// TIA Portal project "Traffic_Light" (V16)

(* hardware
DEVICE "S7-1200 station_1"  S7-1200 Station
   slot 0: "Rack_0"  S7-1200 Rack  Rack  V1.0
   slot 1: "PLC_1"  CPU 1214C DC/DC/DC  6ES7 214-1AG40-0XB0  V4.4
DEVICE "HMI_1"  KTP700 Basic PN
   slot 0: "HMI_1"  KTP700 Basic PN  6AV2 123-2GB03-0AX0  16.0.0.0
   slot 1: "HMI_RT_1"  KTP700 Basic PN  6AV2 123-2GB03-0AX0  16.0.0.0
   slot 5: "HMI_1.IE_CP_1"  PROFINET Interface  16.0.0.0
      slot 1: "PROFINET Interface_1"  PROFINET Interface
         slot 1: "Port_1"  Port
*)

// ===== PLC "PLC_1"  CPU 1214C DC/DC/DC =====

VAR_GLOBAL   // PLC tag table "Default tag table"
   "TrungGian" AT %M10.1 : Bool;
   "Clock_Byte" AT %MB0 : Byte;
   "Clock_10Hz" AT %M0.0 : Bool;
   "Clock_5Hz" AT %M0.1 : Bool;
   "Clock_2.5Hz" AT %M0.2 : Bool;
   "Clock_2Hz" AT %M0.3 : Bool;
   "Clock_1.25Hz" AT %M0.4 : Bool;
   "Clock_1Hz" AT %M0.5 : Bool;
   "Clock_0.625Hz" AT %M0.6 : Bool;
   "Clock_0.5Hz" AT %M0.7 : Bool;
   "Tag_1" AT %M20.1 : Bool;
END_VAR

DATA_BLOCK "DGT_DB"   // DB1
{ S7_Optimized_Access := 'TRUE' }
VERSION : 0.1
   VAR
      SP_TimerXA : Time := T#5S;
      SP_TimerVA : Time := T#3S;
      SP_TimerXB : Time := T#5S;
      SP_TimerVB : Time := T#3S;
      SP_TimerXA_PA4 : Int := 10;
      SP_TimerVA_PA4 : Int := 5;
      SP_TimerXB_PA4 : Int := 10;
      SP_TimerVB_PA4 : Int := 5;
      Lamp_PA1 : Bool;
      Lamp_PA2 : Bool;
      Lamp_PA4 : Bool;
      Update : Bool;
      Update_PA4 : Bool;
      Cancel : Bool;
      Temp_Update : Bool;
      Temp_Update_PA4 : Bool;
      Trunggian_Timer_1 : Bool;
      Trunggian_Timer_2 : Bool;
      OUT_XA : Bool;
      OUT_VA : Bool;
      OUT_DA : Bool;
      OUT_XB : Bool;
      OUT_VB : Bool;
      OUT_DB : Bool;
      OUT_XA_PA2 : Bool;
      OUT_VA_PA2 : Bool;
      OUT_DA_PA2 : Bool;
      OUT_XB_PA2 : Bool;
      OUT_VB_PA2 : Bool;
      OUT_DB_PA2 : Bool;
      OUT_XA_PA3 : Bool;
      OUT_VA_PA3 : Bool;
      OUT_DA_PA3 : Bool;
      OUT_XB_PA3 : Bool;
      OUT_VB_PA3 : Bool;
      OUT_DB_PA3 : Bool;
      OUT_XA_PA4 : Bool;
      OUT_VA_PA4 : Bool;
      OUT_DA_PA4 : Bool;
      OUT_XB_PA4 : Bool;
      OUT_VB_PA4 : Bool;
      OUT_DB_PA4 : Bool;
   END_VAR
BEGIN
END_DATA_BLOCK

DATA_BLOCK "DGT_TempVars"   // DB2
{ S7_Optimized_Access := 'TRUE' }
VERSION : 0.1
   VAR
      T1 : Time := T#5S;
      T2 : Time := T#8S;
      T3 : Time := T#13S;
      T4 : Time := T#16S;
      T1_PA4 : Int := 10;
      T2_PA4 : Int := 15;
      T3_PA4 : Int := 25;
      T4_PA4 : Int := 30;
      Temp : UInt;
      Temp_A : UInt;
      Temp_A_Chuc : UInt;
      Temp_A_DV : UInt;
      Temp_B : UInt;
      Temp_B_Chuc : UInt;
      Temp_B_DV : UInt;
      T11 : UInt;
      T22 : UInt;
      T33 : UInt;
      T44 : UInt;
      Temp_CK_PP1 : Time;
      Temp_SP_XA : Time := T#5S;
      Temp_SP_VA : Time := T#3S;
      Temp_SP_XB : Time := T#5S;
      Temp_SP_VB : Time := T#3S;
   END_VAR
BEGIN
END_DATA_BLOCK

DATA_BLOCK "Control"   // DB4
{ S7_Optimized_Access := 'TRUE' }
VERSION : 0.1
   VAR
      PA1_En : Bool;
      PA2_En : Bool;
      PA3_En : Bool;
      PA4_En : Bool;
      "ON/OFF_PP1" : Bool;
      "ON/OFF_PP2" : Bool;
      "ON/OFF_PP3" : Bool;
      "ON/OFF_PP4" : Bool;
      Stop : Bool;
   END_VAR
BEGIN
END_DATA_BLOCK

DATA_BLOCK "BCD_SEG_TEMPA_CHUC"   // DB10
{ S7_Optimized_Access := 'TRUE' }
VERSION : 0.1
// stored: InstanceOfName BCD_SEG
"BCD_SEG"
BEGIN
END_DATA_BLOCK

DATA_BLOCK "BCD_SEG_TEMPA_DV"   // DB11
{ S7_Optimized_Access := 'TRUE' }
VERSION : 0.1
// stored: InstanceOfName BCD_SEG
"BCD_SEG"
BEGIN
END_DATA_BLOCK

DATA_BLOCK "BCD_SEG_TEMPB_CHUC"   // DB12
{ S7_Optimized_Access := 'TRUE' }
VERSION : 0.1
// stored: InstanceOfName BCD_SEG
"BCD_SEG"
BEGIN
END_DATA_BLOCK

DATA_BLOCK "BCD_SEG_TEMPB_DV"   // DB13
{ S7_Optimized_Access := 'TRUE' }
VERSION : 0.1
// stored: InstanceOfName BCD_SEG
"BCD_SEG"
BEGIN
END_DATA_BLOCK

// folder: System blocks/Program resources

DATA_BLOCK "Timer_PP2"   // DB3
{ S7_Optimized_Access := 'TRUE' }
AUTHOR : Simatic
FAMILY : IEC
NAME : IEC_TMR
VERSION : 1.0
// stored: InstanceOfName IEC_TIMER
"IEC_TIMER"
BEGIN
END_DATA_BLOCK

DATA_BLOCK "T1_TIMER_PP1"   // DB5
{ S7_Optimized_Access := 'TRUE' }
AUTHOR : Simatic
FAMILY : IEC
NAME : IEC_TMR
VERSION : 1.0
// stored: InstanceOfName IEC_TIMER
"IEC_TIMER"
BEGIN
END_DATA_BLOCK

DATA_BLOCK "T2_TIMER_PP1"   // DB6
{ S7_Optimized_Access := 'TRUE' }
AUTHOR : Simatic
FAMILY : IEC
NAME : IEC_TMR
VERSION : 1.0
// stored: InstanceOfName IEC_TIMER
"IEC_TIMER"
BEGIN
END_DATA_BLOCK

DATA_BLOCK "T3_TIMER_PP1"   // DB7
{ S7_Optimized_Access := 'TRUE' }
AUTHOR : Simatic
FAMILY : IEC
NAME : IEC_TMR
VERSION : 1.0
// stored: InstanceOfName IEC_TIMER
"IEC_TIMER"
BEGIN
END_DATA_BLOCK

DATA_BLOCK "T4_TIMER_PP1"   // DB8
{ S7_Optimized_Access := 'TRUE' }
AUTHOR : Simatic
FAMILY : IEC
NAME : IEC_TMR
VERSION : 1.0
// stored: InstanceOfName IEC_TIMER
"IEC_TIMER"
BEGIN
END_DATA_BLOCK

DATA_BLOCK "Timer_PP1"   // DB9
{ S7_Optimized_Access := 'TRUE' }
AUTHOR : Simatic
FAMILY : IEC
NAME : IEC_TMR
VERSION : 1.0
// stored: InstanceOfName IEC_TIMER
"IEC_TIMER"
BEGIN
END_DATA_BLOCK

DATA_BLOCK "C1_PA4"   // DB14
{ S7_Optimized_Access := 'TRUE' }
AUTHOR : Simatic
FAMILY : IEC
NAME : CNTR
VERSION : 1.0
// stored: InstanceOfName IEC_COUNTER
"IEC_COUNTER"
BEGIN
END_DATA_BLOCK

// folder: (top level)

FUNCTION_BLOCK "BCD_SEG"   // FB1, SCL
{ S7_Optimized_Access := 'TRUE' }
VERSION : 0.1
   VAR_INPUT
      BCD : Int;
   END_VAR
   VAR_OUTPUT
      SEG : Byte;
   END_VAR
   VAR_TEMP
      tmp : Byte;
   END_VAR
BEGIN
   IF #BCD = 0 THEN
       // Statement section IF
       #tmp := 63;
   END_IF;
   IF #BCD = 1 THEN
       // Statement section IF
       #tmp := 6;
   END_IF;
   IF #BCD = 2 THEN
       // Statement section IF
       #tmp := 91;
   END_IF;
   IF #BCD = 3 THEN
       // Statement section IF
       #tmp := 79;
   END_IF;
   IF #BCD = 4 THEN
       // Statement section IF
       #tmp := 102;
   END_IF;
   IF #BCD = 5 THEN
       // Statement section IF
       #tmp := 109;
   END_IF;
   IF #BCD = 6 THEN
       // Statement section IF
       #tmp := 125;
   END_IF;
   IF #BCD = 7 THEN
       // Statement section IF
       #tmp := 7;
   END_IF;
   IF #BCD = 8 THEN
       // Statement section IF
       #tmp := 127;
   END_IF;
   IF #BCD = 9 THEN
       // Statement section IF
       #tmp := 111;
   END_IF;
   #SEG := #tmp;
END_FUNCTION_BLOCK

FUNCTION "PA2" : Void   // FC1, LAD
{ S7_Optimized_Access := 'TRUE' }
VERSION : 0.1
   VAR_INPUT
      EN_2 : Bool;
   END_VAR
   VAR_TEMP   // added for the SCL form of the ladder/FBD networks
      _w1 : Bool;
      _w2 : Bool;
   END_VAR
BEGIN

REGION Network 1: Update
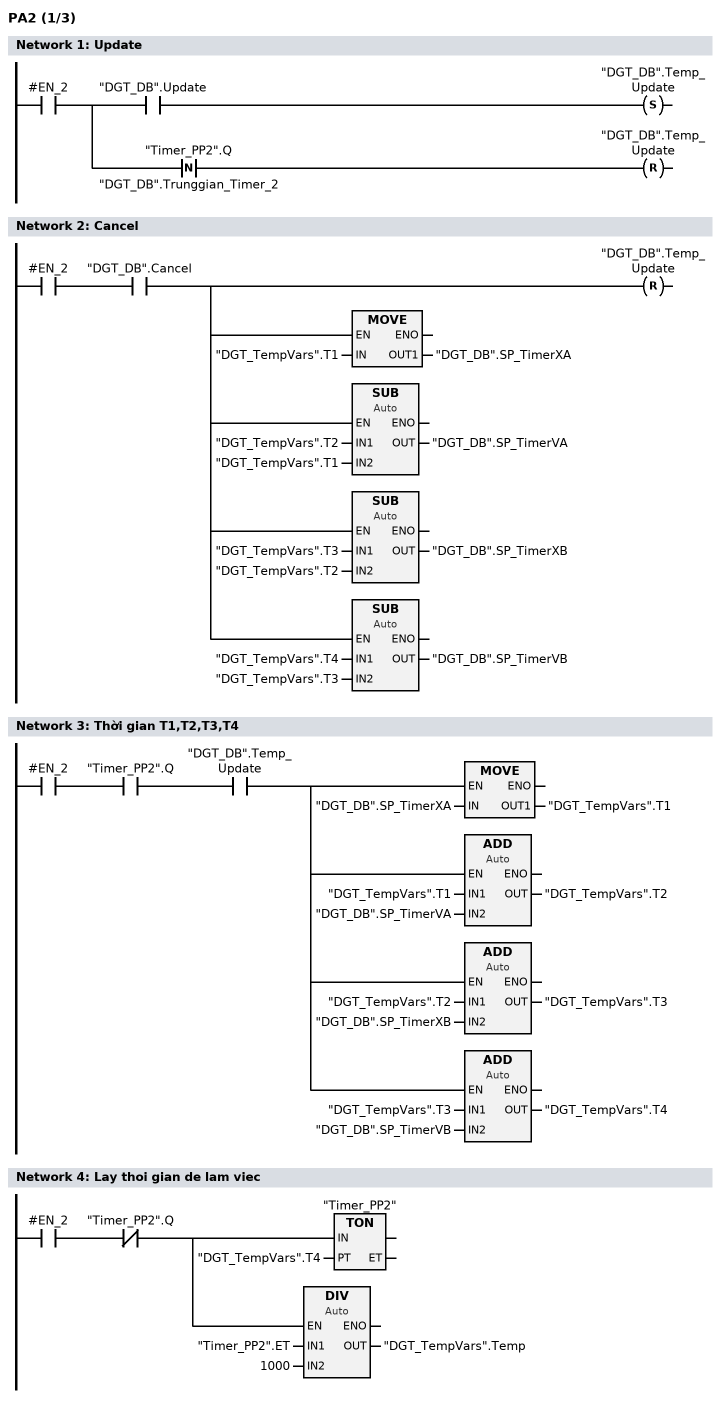
   RUNG wire#powerrail
      Contact( #EN_2 )
      wire#w1
      Contact( "DGT_DB".Update )
      S_Coil( "DGT_DB".Temp_Update )
   END_RUNG
   RUNG wire#w1
      N_Contact(operand := "Timer_PP2".Q, bit := "DGT_DB".Trunggian_Timer_2)
      R_Coil( "DGT_DB".Temp_Update )
   END_RUNG
   // the same network as SCL:
   IF #EN_2 AND "DGT_DB".Update THEN "DGT_DB".Temp_Update := TRUE; END_IF;
   #_w1 := #EN_2 AND NOT "Timer_PP2".Q AND "DGT_DB".Trunggian_Timer_2;   // falling edge of "Timer_PP2".Q
   "DGT_DB".Trunggian_Timer_2 := "Timer_PP2".Q;
   IF #_w1 THEN "DGT_DB".Temp_Update := FALSE; END_IF;
END_REGION

REGION Network 2: Cancel
   RUNG wire#powerrail
      Contact( #EN_2 )
      Contact( "DGT_DB".Cancel )
      wire#w1
      R_Coil( "DGT_DB".Temp_Update )
   END_RUNG
   RUNG wire#w1
      Move(in := "DGT_TempVars".T1, out1 => "DGT_DB".SP_TimerXA)
   END_RUNG
   RUNG wire#w1
      Sub(in1 := "DGT_TempVars".T2, in2 := "DGT_TempVars".T1, out => "DGT_DB".SP_TimerVA)
   END_RUNG
   RUNG wire#w1
      Sub(in1 := "DGT_TempVars".T3, in2 := "DGT_TempVars".T2, out => "DGT_DB".SP_TimerXB)
   END_RUNG
   RUNG wire#w1
      Sub(in1 := "DGT_TempVars".T4, in2 := "DGT_TempVars".T3, out => "DGT_DB".SP_TimerVB)
   END_RUNG
   // the same network as SCL:
   IF #EN_2 AND "DGT_DB".Cancel THEN
       "DGT_DB".Temp_Update := FALSE;
       "DGT_DB".SP_TimerXA := "DGT_TempVars".T1;
       "DGT_DB".SP_TimerVA := "DGT_TempVars".T2 - "DGT_TempVars".T1;
       "DGT_DB".SP_TimerXB := "DGT_TempVars".T3 - "DGT_TempVars".T2;
       "DGT_DB".SP_TimerVB := "DGT_TempVars".T4 - "DGT_TempVars".T3;
   END_IF;
END_REGION

REGION Network 3: Thời gian T1,T2,T3,T4
   RUNG wire#powerrail
      Contact( #EN_2 )
      Contact( "Timer_PP2".Q )
      Contact( "DGT_DB".Temp_Update )
      wire#w1
      Move(in := "DGT_DB".SP_TimerXA, out1 => "DGT_TempVars".T1)
   END_RUNG
   RUNG wire#w1
      Add(in1 := "DGT_TempVars".T1, in2 := "DGT_DB".SP_TimerVA, out => "DGT_TempVars".T2)
   END_RUNG
   RUNG wire#w1
      Add(in1 := "DGT_TempVars".T2, in2 := "DGT_DB".SP_TimerXB, out => "DGT_TempVars".T3)
   END_RUNG
   RUNG wire#w1
      Add(in1 := "DGT_TempVars".T3, in2 := "DGT_DB".SP_TimerVB, out => "DGT_TempVars".T4)
   END_RUNG
   // the same network as SCL:
   IF #EN_2 AND "Timer_PP2".Q AND "DGT_DB".Temp_Update THEN
       "DGT_TempVars".T1 := "DGT_DB".SP_TimerXA;
       "DGT_TempVars".T2 := "DGT_TempVars".T1 + "DGT_DB".SP_TimerVA;
       "DGT_TempVars".T3 := "DGT_TempVars".T2 + "DGT_DB".SP_TimerXB;
       "DGT_TempVars".T4 := "DGT_TempVars".T3 + "DGT_DB".SP_TimerVB;
   END_IF;
END_REGION

REGION Network 4: Lay thoi gian de lam viec
   #_w1 := #EN_2 AND NOT "Timer_PP2".Q;
   "Timer_PP2".TON(IN := #_w1, PT := "DGT_TempVars".T4);
   IF #_w1 THEN "DGT_TempVars".Temp := "Timer_PP2".ET / 1000; END_IF;
END_REGION

REGION Network 5: XA,VA,XB,VB
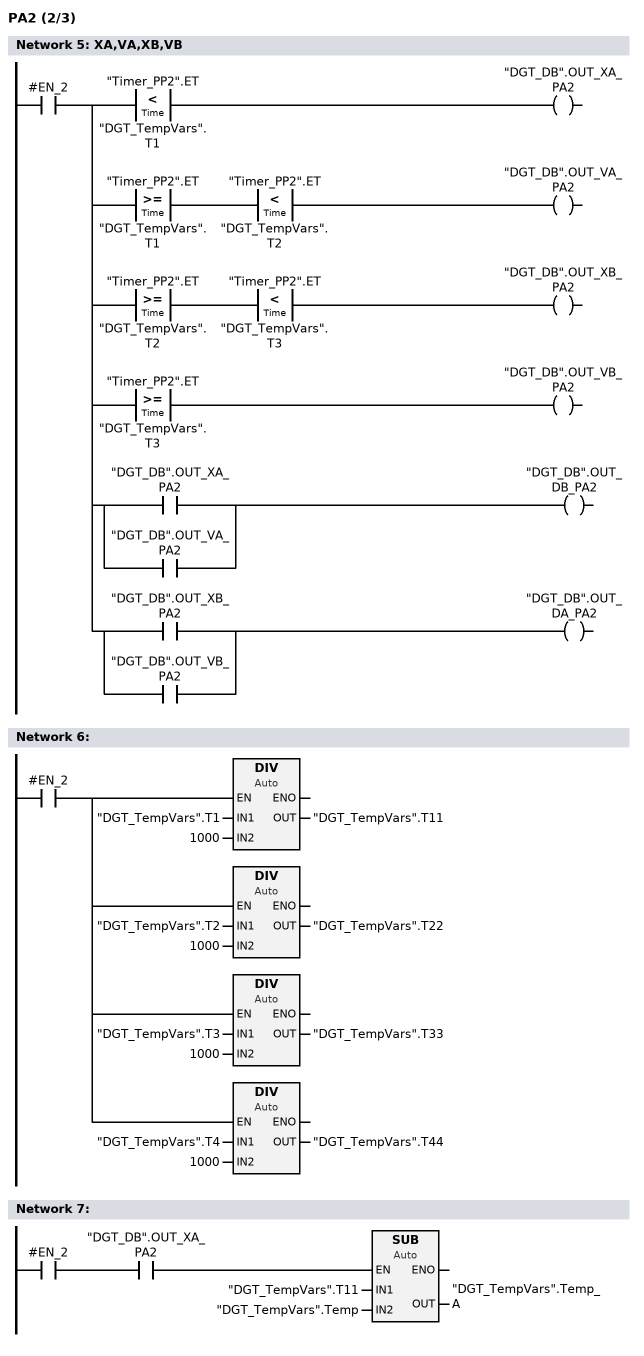
   RUNG wire#powerrail
      Contact( #EN_2 )
      wire#w1
      { S7_Templates := "SrcType := Time" } LT_Contact(in1 := "Timer_PP2".ET, in2 := "DGT_TempVars".T1)
      Coil( "DGT_DB".OUT_XA_PA2 )
   END_RUNG
   RUNG wire#w1
      { S7_Templates := "SrcType := Time" } GE_Contact(in1 := "Timer_PP2".ET, in2 := "DGT_TempVars".T1)
      { S7_Templates := "SrcType := Time" } LT_Contact(in1 := "Timer_PP2".ET, in2 := "DGT_TempVars".T2)
      Coil( "DGT_DB".OUT_VA_PA2 )
   END_RUNG
   RUNG wire#w1
      { S7_Templates := "SrcType := Time" } GE_Contact(in1 := "Timer_PP2".ET, in2 := "DGT_TempVars".T2)
      { S7_Templates := "SrcType := Time" } LT_Contact(in1 := "Timer_PP2".ET, in2 := "DGT_TempVars".T3)
      Coil( "DGT_DB".OUT_XB_PA2 )
   END_RUNG
   RUNG wire#w1
      { S7_Templates := "SrcType := Time" } GE_Contact(in1 := "Timer_PP2".ET, in2 := "DGT_TempVars".T3)
      Coil( "DGT_DB".OUT_VB_PA2 )
   END_RUNG
   RUNG wire#w1
      Contact( "DGT_DB".OUT_XA_PA2 )
      wire#w2
      Coil( "DGT_DB".OUT_DB_PA2 )
   END_RUNG
   RUNG wire#w1
      Contact( "DGT_DB".OUT_VA_PA2 )
   END_RUNG wire#w2
   RUNG wire#w1
      Contact( "DGT_DB".OUT_XB_PA2 )
      wire#w3
      Coil( "DGT_DB".OUT_DA_PA2 )
   END_RUNG
   RUNG wire#w1
      Contact( "DGT_DB".OUT_VB_PA2 )
   END_RUNG wire#w3
   // the same network as SCL:
   "DGT_DB".OUT_XA_PA2 := #EN_2 AND ("Timer_PP2".ET < "DGT_TempVars".T1);
   "DGT_DB".OUT_VA_PA2 := #EN_2 AND ("Timer_PP2".ET >= "DGT_TempVars".T1) AND ("Timer_PP2".ET < "DGT_TempVars".T2);
   "DGT_DB".OUT_XB_PA2 := #EN_2 AND ("Timer_PP2".ET >= "DGT_TempVars".T2) AND ("Timer_PP2".ET < "DGT_TempVars".T3);
   "DGT_DB".OUT_VB_PA2 := #EN_2 AND ("Timer_PP2".ET >= "DGT_TempVars".T3);
   "DGT_DB".OUT_DB_PA2 := #EN_2 AND ("DGT_DB".OUT_XA_PA2 OR "DGT_DB".OUT_VA_PA2);
   "DGT_DB".OUT_DA_PA2 := #EN_2 AND ("DGT_DB".OUT_XB_PA2 OR "DGT_DB".OUT_VB_PA2);
END_REGION

REGION Network 6
   RUNG wire#powerrail
      Contact( #EN_2 )
      wire#w1
      Div(in1 := "DGT_TempVars".T1, in2 := 1000, out => "DGT_TempVars".T11)
   END_RUNG
   RUNG wire#w1
      Div(in1 := "DGT_TempVars".T2, in2 := 1000, out => "DGT_TempVars".T22)
   END_RUNG
   RUNG wire#w1
      Div(in1 := "DGT_TempVars".T3, in2 := 1000, out => "DGT_TempVars".T33)
   END_RUNG
   RUNG wire#w1
      Div(in1 := "DGT_TempVars".T4, in2 := 1000, out => "DGT_TempVars".T44)
   END_RUNG
   // the same network as SCL:
   IF #EN_2 THEN
       "DGT_TempVars".T11 := "DGT_TempVars".T1 / 1000;
       "DGT_TempVars".T22 := "DGT_TempVars".T2 / 1000;
       "DGT_TempVars".T33 := "DGT_TempVars".T3 / 1000;
       "DGT_TempVars".T44 := "DGT_TempVars".T4 / 1000;
   END_IF;
END_REGION

REGION Network 7
   RUNG wire#powerrail
      Contact( #EN_2 )
      Contact( "DGT_DB".OUT_XA_PA2 )
      Sub(in1 := "DGT_TempVars".T11, in2 := "DGT_TempVars".Temp, out => "DGT_TempVars".Temp_A)
   END_RUNG
   // the same network as SCL:
   IF #EN_2 AND "DGT_DB".OUT_XA_PA2 THEN
       "DGT_TempVars".Temp_A := "DGT_TempVars".T11 - "DGT_TempVars".Temp;
   END_IF;
END_REGION

REGION Network 8
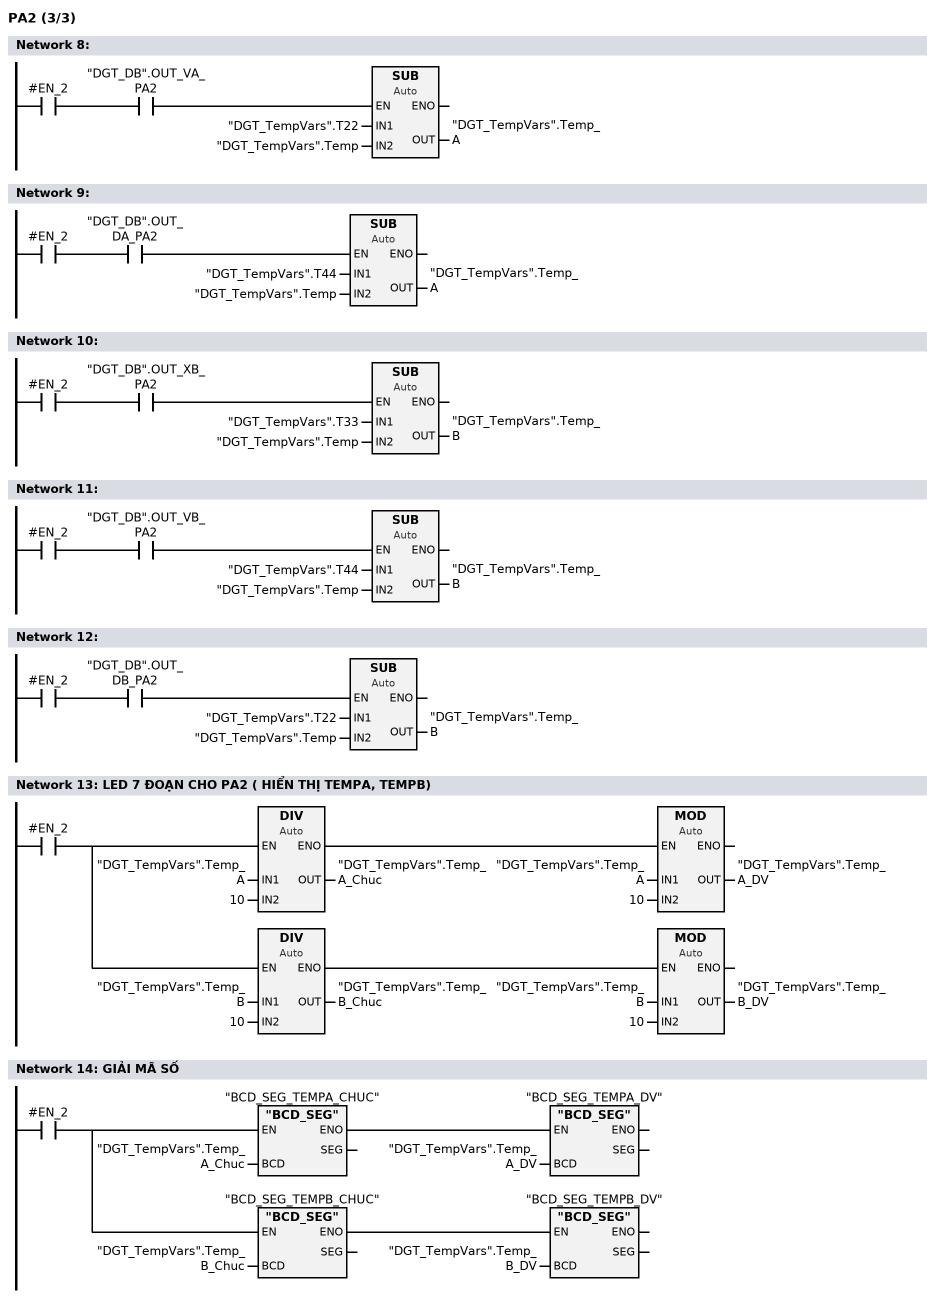
   RUNG wire#powerrail
      Contact( #EN_2 )
      Contact( "DGT_DB".OUT_VA_PA2 )
      Sub(in1 := "DGT_TempVars".T22, in2 := "DGT_TempVars".Temp, out => "DGT_TempVars".Temp_A)
   END_RUNG
   // the same network as SCL:
   IF #EN_2 AND "DGT_DB".OUT_VA_PA2 THEN
       "DGT_TempVars".Temp_A := "DGT_TempVars".T22 - "DGT_TempVars".Temp;
   END_IF;
END_REGION

REGION Network 9
   RUNG wire#powerrail
      Contact( #EN_2 )
      Contact( "DGT_DB".OUT_DA_PA2 )
      Sub(in1 := "DGT_TempVars".T44, in2 := "DGT_TempVars".Temp, out => "DGT_TempVars".Temp_A)
   END_RUNG
   // the same network as SCL:
   IF #EN_2 AND "DGT_DB".OUT_DA_PA2 THEN
       "DGT_TempVars".Temp_A := "DGT_TempVars".T44 - "DGT_TempVars".Temp;
   END_IF;
END_REGION

REGION Network 10
   RUNG wire#powerrail
      Contact( #EN_2 )
      Contact( "DGT_DB".OUT_XB_PA2 )
      Sub(in1 := "DGT_TempVars".T33, in2 := "DGT_TempVars".Temp, out => "DGT_TempVars".Temp_B)
   END_RUNG
   // the same network as SCL:
   IF #EN_2 AND "DGT_DB".OUT_XB_PA2 THEN
       "DGT_TempVars".Temp_B := "DGT_TempVars".T33 - "DGT_TempVars".Temp;
   END_IF;
END_REGION

REGION Network 11
   RUNG wire#powerrail
      Contact( #EN_2 )
      Contact( "DGT_DB".OUT_VB_PA2 )
      Sub(in1 := "DGT_TempVars".T44, in2 := "DGT_TempVars".Temp, out => "DGT_TempVars".Temp_B)
   END_RUNG
   // the same network as SCL:
   IF #EN_2 AND "DGT_DB".OUT_VB_PA2 THEN
       "DGT_TempVars".Temp_B := "DGT_TempVars".T44 - "DGT_TempVars".Temp;
   END_IF;
END_REGION

REGION Network 12
   RUNG wire#powerrail
      Contact( #EN_2 )
      Contact( "DGT_DB".OUT_DB_PA2 )
      Sub(in1 := "DGT_TempVars".T22, in2 := "DGT_TempVars".Temp, out => "DGT_TempVars".Temp_B)
   END_RUNG
   // the same network as SCL:
   IF #EN_2 AND "DGT_DB".OUT_DB_PA2 THEN
       "DGT_TempVars".Temp_B := "DGT_TempVars".T22 - "DGT_TempVars".Temp;
   END_IF;
END_REGION

REGION Network 13: LED 7 ĐOẠN CHO PA2 ( HIỂN THỊ TEMPA, TEMPB)
   RUNG wire#powerrail
      Contact( #EN_2 )
      wire#w1
      Div(in1 := "DGT_TempVars".Temp_A, in2 := 10, out => "DGT_TempVars".Temp_A_Chuc)
      Mod(in1 := "DGT_TempVars".Temp_A, in2 := 10, out => "DGT_TempVars".Temp_A_DV)
   END_RUNG
   RUNG wire#w1
      Div(in1 := "DGT_TempVars".Temp_B, in2 := 10, out => "DGT_TempVars".Temp_B_Chuc)
      Mod(in1 := "DGT_TempVars".Temp_B, in2 := 10, out => "DGT_TempVars".Temp_B_DV)
   END_RUNG
   // the same network as SCL:
   IF #EN_2 THEN
       "DGT_TempVars".Temp_A_Chuc := "DGT_TempVars".Temp_A / 10;
       "DGT_TempVars".Temp_A_DV := "DGT_TempVars".Temp_A MOD 10;
       "DGT_TempVars".Temp_B_Chuc := "DGT_TempVars".Temp_B / 10;
       "DGT_TempVars".Temp_B_DV := "DGT_TempVars".Temp_B MOD 10;
   END_IF;
END_REGION

REGION Network 14: GIẢI MÃ SỐ
   RUNG wire#powerrail
      Contact( #EN_2 )
      wire#w1
      "BCD_SEG_TEMPA_CHUC"(BCD := "DGT_TempVars".Temp_A_Chuc, SEG =>)
      "BCD_SEG_TEMPA_DV"(BCD := "DGT_TempVars".Temp_A_DV, SEG =>)
   END_RUNG
   RUNG wire#w1
      "BCD_SEG_TEMPB_CHUC"(BCD := "DGT_TempVars".Temp_B_Chuc, SEG =>)
      "BCD_SEG_TEMPB_DV"(BCD := "DGT_TempVars".Temp_B_DV, SEG =>)
   END_RUNG
   // the same network as SCL:
   "BCD_SEG_TEMPA_CHUC"(EN := #EN_2, BCD := "DGT_TempVars".Temp_A_Chuc, ENO => #_w1);   // "BCD_SEG"
   IF #_w1 THEN
       "BCD_SEG_TEMPA_DV"(BCD := "DGT_TempVars".Temp_A_DV);   // "BCD_SEG"
   END_IF;
   "BCD_SEG_TEMPB_CHUC"(EN := #EN_2, BCD := "DGT_TempVars".Temp_B_Chuc, ENO => #_w2);   // "BCD_SEG"
   IF #_w2 THEN
       "BCD_SEG_TEMPB_DV"(BCD := "DGT_TempVars".Temp_B_DV);   // "BCD_SEG"
   END_IF;
END_REGION
END_FUNCTION

FUNCTION "PA1" : Void   // FC2, LAD
{ S7_Optimized_Access := 'TRUE' }
VERSION : 0.1
   VAR_INPUT
      EN_1 : Bool;
   END_VAR
   VAR_TEMP   // added for the SCL form of the ladder/FBD networks
      _w1 : Bool;
      _w2 : Bool;
      _w3 : Bool;
   END_VAR
BEGIN

REGION Network 1: Update
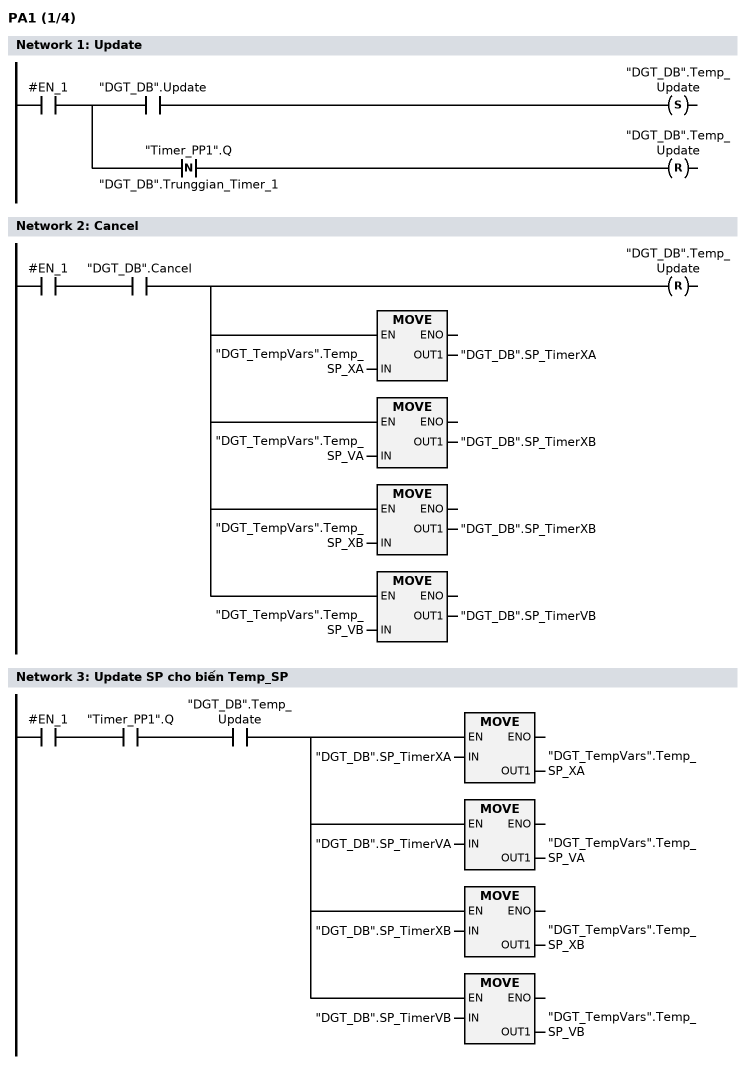
   RUNG wire#powerrail
      Contact( #EN_1 )
      wire#w1
      Contact( "DGT_DB".Update )
      S_Coil( "DGT_DB".Temp_Update )
   END_RUNG
   RUNG wire#w1
      N_Contact(operand := "Timer_PP1".Q, bit := "DGT_DB".Trunggian_Timer_1)
      R_Coil( "DGT_DB".Temp_Update )
   END_RUNG
   // the same network as SCL:
   IF #EN_1 AND "DGT_DB".Update THEN "DGT_DB".Temp_Update := TRUE; END_IF;
   #_w1 := #EN_1 AND NOT "Timer_PP1".Q AND "DGT_DB".Trunggian_Timer_1;   // falling edge of "Timer_PP1".Q
   "DGT_DB".Trunggian_Timer_1 := "Timer_PP1".Q;
   IF #_w1 THEN "DGT_DB".Temp_Update := FALSE; END_IF;
END_REGION

REGION Network 2: Cancel
   RUNG wire#powerrail
      Contact( #EN_1 )
      Contact( "DGT_DB".Cancel )
      wire#w1
      R_Coil( "DGT_DB".Temp_Update )
   END_RUNG
   RUNG wire#w1
      Move(in := "DGT_TempVars".Temp_SP_XA, out1 => "DGT_DB".SP_TimerXA)
   END_RUNG
   RUNG wire#w1
      Move(in := "DGT_TempVars".Temp_SP_VA, out1 => "DGT_DB".SP_TimerXB)
   END_RUNG
   RUNG wire#w1
      Move(in := "DGT_TempVars".Temp_SP_XB, out1 => "DGT_DB".SP_TimerXB)
   END_RUNG
   RUNG wire#w1
      Move(in := "DGT_TempVars".Temp_SP_VB, out1 => "DGT_DB".SP_TimerVB)
   END_RUNG
   // the same network as SCL:
   IF #EN_1 AND "DGT_DB".Cancel THEN
       "DGT_DB".Temp_Update := FALSE;
       "DGT_DB".SP_TimerXA := "DGT_TempVars".Temp_SP_XA;
       "DGT_DB".SP_TimerXB := "DGT_TempVars".Temp_SP_VA;
       "DGT_DB".SP_TimerXB := "DGT_TempVars".Temp_SP_XB;
       "DGT_DB".SP_TimerVB := "DGT_TempVars".Temp_SP_VB;
   END_IF;
END_REGION

REGION Network 3: Update SP cho biến Temp_SP
   RUNG wire#powerrail
      Contact( #EN_1 )
      Contact( "Timer_PP1".Q )
      Contact( "DGT_DB".Temp_Update )
      wire#w1
      Move(in := "DGT_DB".SP_TimerXA, out1 => "DGT_TempVars".Temp_SP_XA)
   END_RUNG
   RUNG wire#w1
      Move(in := "DGT_DB".SP_TimerVA, out1 => "DGT_TempVars".Temp_SP_VA)
   END_RUNG
   RUNG wire#w1
      Move(in := "DGT_DB".SP_TimerXB, out1 => "DGT_TempVars".Temp_SP_XB)
   END_RUNG
   RUNG wire#w1
      Move(in := "DGT_DB".SP_TimerVB, out1 => "DGT_TempVars".Temp_SP_VB)
   END_RUNG
   // the same network as SCL:
   IF #EN_1 AND "Timer_PP1".Q AND "DGT_DB".Temp_Update THEN
       "DGT_TempVars".Temp_SP_XA := "DGT_DB".SP_TimerXA;
       "DGT_TempVars".Temp_SP_VA := "DGT_DB".SP_TimerVA;
       "DGT_TempVars".Temp_SP_XB := "DGT_DB".SP_TimerXB;
       "DGT_TempVars".Temp_SP_VB := "DGT_DB".SP_TimerVB;
   END_IF;
END_REGION

REGION Network 4: Den Giao Thong
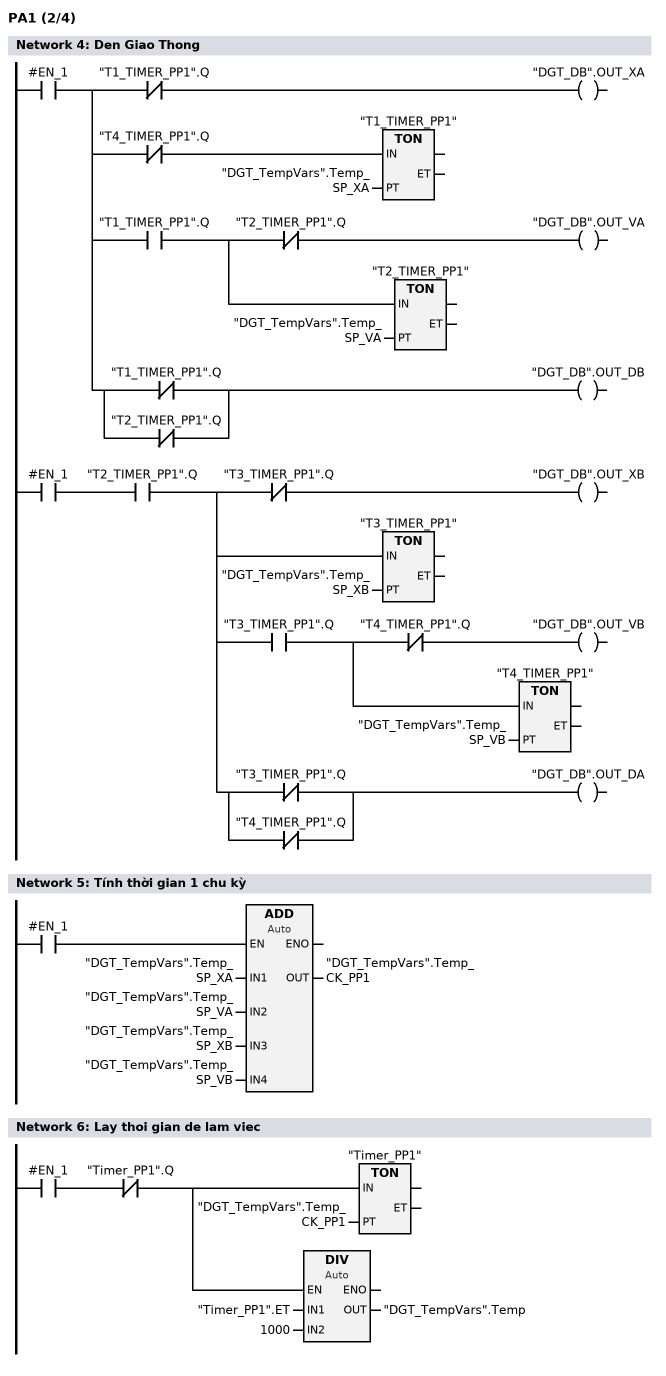
   "DGT_DB".OUT_XA := #EN_1 AND NOT "T1_TIMER_PP1".Q;
   "T1_TIMER_PP1".TON(IN := #EN_1 AND NOT "T4_TIMER_PP1".Q, PT := "DGT_TempVars".Temp_SP_XA);
   #_w1 := #EN_1 AND "T1_TIMER_PP1".Q;
   "DGT_DB".OUT_VA := #_w1 AND NOT "T2_TIMER_PP1".Q;
   "T2_TIMER_PP1".TON(IN := #_w1, PT := "DGT_TempVars".Temp_SP_VA);
   "DGT_DB".OUT_DB := #EN_1 AND (NOT "T1_TIMER_PP1".Q OR NOT "T2_TIMER_PP1".Q);
   #_w2 := #EN_1 AND "T2_TIMER_PP1".Q;
   "DGT_DB".OUT_XB := #_w2 AND NOT "T3_TIMER_PP1".Q;
   "T3_TIMER_PP1".TON(IN := #_w2, PT := "DGT_TempVars".Temp_SP_XB);
   #_w3 := #_w2 AND "T3_TIMER_PP1".Q;
   "DGT_DB".OUT_VB := #_w3 AND NOT "T4_TIMER_PP1".Q;
   "T4_TIMER_PP1".TON(IN := #_w3, PT := "DGT_TempVars".Temp_SP_VB);
   "DGT_DB".OUT_DA := #_w2 AND (NOT "T3_TIMER_PP1".Q OR NOT "T4_TIMER_PP1".Q);
END_REGION

REGION Network 5: Tính thời gian 1 chu kỳ
   RUNG wire#powerrail
      Contact( #EN_1 )
      Add(in1 := "DGT_TempVars".Temp_SP_XA, in2 := "DGT_TempVars".Temp_SP_VA, in3 := "DGT_TempVars".Temp_SP_XB, in4 := "DGT_TempVars".Temp_SP_VB, out => "DGT_TempVars".Temp_CK_PP1)
   END_RUNG
   // the same network as SCL:
   IF #EN_1 THEN
       "DGT_TempVars".Temp_CK_PP1 := "DGT_TempVars".Temp_SP_XA + "DGT_TempVars".Temp_SP_VA + "DGT_TempVars".Temp_SP_XB + "DGT_TempVars".Temp_SP_VB;
   END_IF;
END_REGION

REGION Network 6: Lay thoi gian de lam viec
   #_w1 := #EN_1 AND NOT "Timer_PP1".Q;
   "Timer_PP1".TON(IN := #_w1, PT := "DGT_TempVars".Temp_CK_PP1);
   IF #_w1 THEN "DGT_TempVars".Temp := "Timer_PP1".ET / 1000; END_IF;
END_REGION

REGION Network 7: Thời gian T1,T2,T3,T4
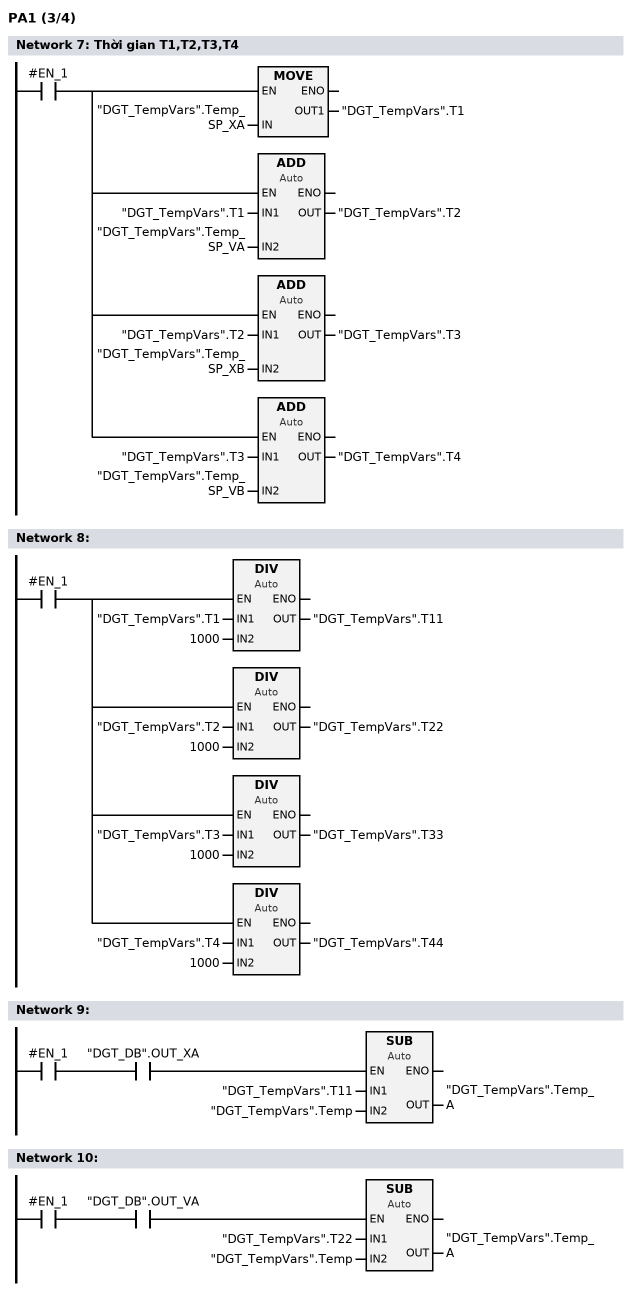
   RUNG wire#powerrail
      Contact( #EN_1 )
      wire#w1
      Move(in := "DGT_TempVars".Temp_SP_XA, out1 => "DGT_TempVars".T1)
   END_RUNG
   RUNG wire#w1
      Add(in1 := "DGT_TempVars".T1, in2 := "DGT_TempVars".Temp_SP_VA, out => "DGT_TempVars".T2)
   END_RUNG
   RUNG wire#w1
      Add(in1 := "DGT_TempVars".T2, in2 := "DGT_TempVars".Temp_SP_XB, out => "DGT_TempVars".T3)
   END_RUNG
   RUNG wire#w1
      Add(in1 := "DGT_TempVars".T3, in2 := "DGT_TempVars".Temp_SP_VB, out => "DGT_TempVars".T4)
   END_RUNG
   // the same network as SCL:
   IF #EN_1 THEN
       "DGT_TempVars".T1 := "DGT_TempVars".Temp_SP_XA;
       "DGT_TempVars".T2 := "DGT_TempVars".T1 + "DGT_TempVars".Temp_SP_VA;
       "DGT_TempVars".T3 := "DGT_TempVars".T2 + "DGT_TempVars".Temp_SP_XB;
       "DGT_TempVars".T4 := "DGT_TempVars".T3 + "DGT_TempVars".Temp_SP_VB;
   END_IF;
END_REGION

REGION Network 8
   RUNG wire#powerrail
      Contact( #EN_1 )
      wire#w1
      Div(in1 := "DGT_TempVars".T1, in2 := 1000, out => "DGT_TempVars".T11)
   END_RUNG
   RUNG wire#w1
      Div(in1 := "DGT_TempVars".T2, in2 := 1000, out => "DGT_TempVars".T22)
   END_RUNG
   RUNG wire#w1
      Div(in1 := "DGT_TempVars".T3, in2 := 1000, out => "DGT_TempVars".T33)
   END_RUNG
   RUNG wire#w1
      Div(in1 := "DGT_TempVars".T4, in2 := 1000, out => "DGT_TempVars".T44)
   END_RUNG
   // the same network as SCL:
   IF #EN_1 THEN
       "DGT_TempVars".T11 := "DGT_TempVars".T1 / 1000;
       "DGT_TempVars".T22 := "DGT_TempVars".T2 / 1000;
       "DGT_TempVars".T33 := "DGT_TempVars".T3 / 1000;
       "DGT_TempVars".T44 := "DGT_TempVars".T4 / 1000;
   END_IF;
END_REGION

REGION Network 9
   RUNG wire#powerrail
      Contact( #EN_1 )
      Contact( "DGT_DB".OUT_XA )
      Sub(in1 := "DGT_TempVars".T11, in2 := "DGT_TempVars".Temp, out => "DGT_TempVars".Temp_A)
   END_RUNG
   // the same network as SCL:
   IF #EN_1 AND "DGT_DB".OUT_XA THEN
       "DGT_TempVars".Temp_A := "DGT_TempVars".T11 - "DGT_TempVars".Temp;
   END_IF;
END_REGION

REGION Network 10
   RUNG wire#powerrail
      Contact( #EN_1 )
      Contact( "DGT_DB".OUT_VA )
      Sub(in1 := "DGT_TempVars".T22, in2 := "DGT_TempVars".Temp, out => "DGT_TempVars".Temp_A)
   END_RUNG
   // the same network as SCL:
   IF #EN_1 AND "DGT_DB".OUT_VA THEN
       "DGT_TempVars".Temp_A := "DGT_TempVars".T22 - "DGT_TempVars".Temp;
   END_IF;
END_REGION

REGION Network 11
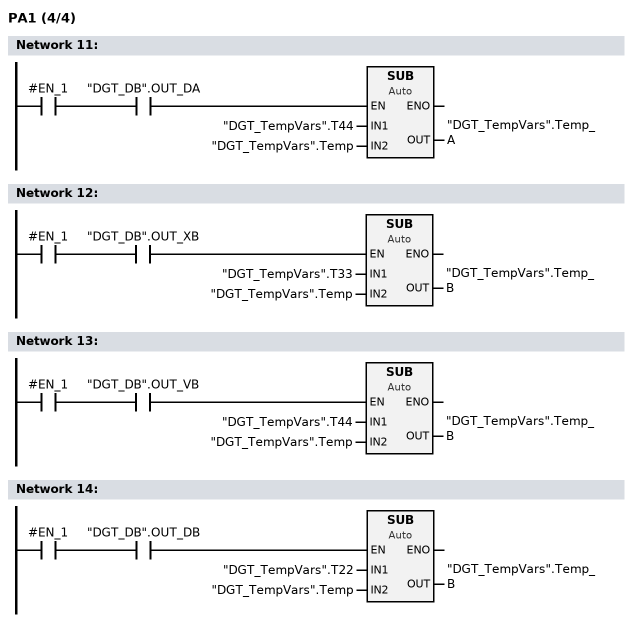
   RUNG wire#powerrail
      Contact( #EN_1 )
      Contact( "DGT_DB".OUT_DA )
      Sub(in1 := "DGT_TempVars".T44, in2 := "DGT_TempVars".Temp, out => "DGT_TempVars".Temp_A)
   END_RUNG
   // the same network as SCL:
   IF #EN_1 AND "DGT_DB".OUT_DA THEN
       "DGT_TempVars".Temp_A := "DGT_TempVars".T44 - "DGT_TempVars".Temp;
   END_IF;
END_REGION

REGION Network 12
   RUNG wire#powerrail
      Contact( #EN_1 )
      Contact( "DGT_DB".OUT_XB )
      Sub(in1 := "DGT_TempVars".T33, in2 := "DGT_TempVars".Temp, out => "DGT_TempVars".Temp_B)
   END_RUNG
   // the same network as SCL:
   IF #EN_1 AND "DGT_DB".OUT_XB THEN
       "DGT_TempVars".Temp_B := "DGT_TempVars".T33 - "DGT_TempVars".Temp;
   END_IF;
END_REGION

REGION Network 13
   RUNG wire#powerrail
      Contact( #EN_1 )
      Contact( "DGT_DB".OUT_VB )
      Sub(in1 := "DGT_TempVars".T44, in2 := "DGT_TempVars".Temp, out => "DGT_TempVars".Temp_B)
   END_RUNG
   // the same network as SCL:
   IF #EN_1 AND "DGT_DB".OUT_VB THEN
       "DGT_TempVars".Temp_B := "DGT_TempVars".T44 - "DGT_TempVars".Temp;
   END_IF;
END_REGION

REGION Network 14
   RUNG wire#powerrail
      Contact( #EN_1 )
      Contact( "DGT_DB".OUT_DB )
      Sub(in1 := "DGT_TempVars".T22, in2 := "DGT_TempVars".Temp, out => "DGT_TempVars".Temp_B)
   END_RUNG
   // the same network as SCL:
   IF #EN_1 AND "DGT_DB".OUT_DB THEN
       "DGT_TempVars".Temp_B := "DGT_TempVars".T22 - "DGT_TempVars".Temp;
   END_IF;
END_REGION
END_FUNCTION

FUNCTION "PA3" : Void   // FC3, LAD
{ S7_Optimized_Access := 'TRUE' }
VERSION : 0.1
BEGIN
END_FUNCTION

FUNCTION "PA4" : Void   // FC4, LAD
{ S7_Optimized_Access := 'TRUE' }
VERSION : 0.1
   VAR_INPUT
      EN_4 : Bool;
   END_VAR
   VAR_TEMP   // added for the SCL form of the ladder/FBD networks
      _w1 : Bool;
      _w2 : Bool;
   END_VAR
BEGIN

REGION Network 1
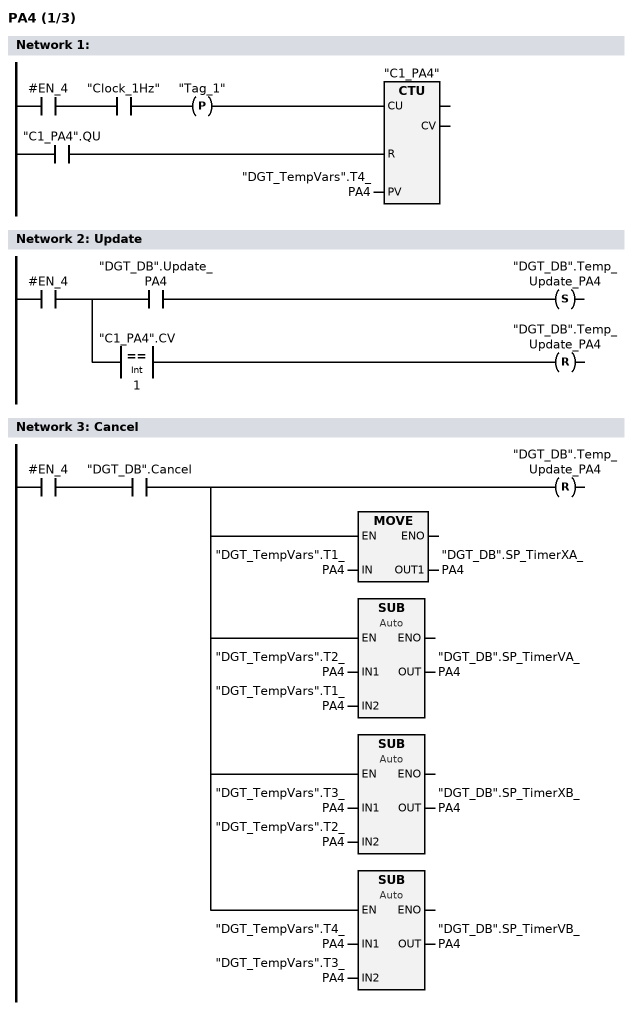
   #_w1 := #EN_4 AND "Clock_1Hz";
   #_w2 := #_w1 AND NOT "Tag_1";   // rising edge
   "Tag_1" := #_w1;
   "C1_PA4".CTU(CU := #_w2, R := "C1_PA4".QU, PV := "DGT_TempVars".T4_PA4);
END_REGION

REGION Network 2: Update
   RUNG wire#powerrail
      Contact( #EN_4 )
      wire#w1
      Contact( "DGT_DB".Update_PA4 )
      S_Coil( "DGT_DB".Temp_Update_PA4 )
   END_RUNG
   RUNG wire#w1
      { S7_Templates := "SrcType := Int" } EQ_Contact(in1 := "C1_PA4".CV, in2 := 1)
      R_Coil( "DGT_DB".Temp_Update_PA4 )
   END_RUNG
   // the same network as SCL:
   IF #EN_4 AND "DGT_DB".Update_PA4 THEN "DGT_DB".Temp_Update_PA4 := TRUE; END_IF;
   IF #EN_4 AND ("C1_PA4".CV = 1) THEN "DGT_DB".Temp_Update_PA4 := FALSE; END_IF;
END_REGION

REGION Network 3: Cancel
   RUNG wire#powerrail
      Contact( #EN_4 )
      Contact( "DGT_DB".Cancel )
      wire#w1
      R_Coil( "DGT_DB".Temp_Update_PA4 )
   END_RUNG
   RUNG wire#w1
      Move(in := "DGT_TempVars".T1_PA4, out1 => "DGT_DB".SP_TimerXA_PA4)
   END_RUNG
   RUNG wire#w1
      Sub(in1 := "DGT_TempVars".T2_PA4, in2 := "DGT_TempVars".T1_PA4, out => "DGT_DB".SP_TimerVA_PA4)
   END_RUNG
   RUNG wire#w1
      Sub(in1 := "DGT_TempVars".T3_PA4, in2 := "DGT_TempVars".T2_PA4, out => "DGT_DB".SP_TimerXB_PA4)
   END_RUNG
   RUNG wire#w1
      Sub(in1 := "DGT_TempVars".T4_PA4, in2 := "DGT_TempVars".T3_PA4, out => "DGT_DB".SP_TimerVB_PA4)
   END_RUNG
   // the same network as SCL:
   IF #EN_4 AND "DGT_DB".Cancel THEN
       "DGT_DB".Temp_Update_PA4 := FALSE;
       "DGT_DB".SP_TimerXA_PA4 := "DGT_TempVars".T1_PA4;
       "DGT_DB".SP_TimerVA_PA4 := "DGT_TempVars".T2_PA4 - "DGT_TempVars".T1_PA4;
       "DGT_DB".SP_TimerXB_PA4 := "DGT_TempVars".T3_PA4 - "DGT_TempVars".T2_PA4;
       "DGT_DB".SP_TimerVB_PA4 := "DGT_TempVars".T4_PA4 - "DGT_TempVars".T3_PA4;
   END_IF;
END_REGION

REGION Network 4: Thời gian T1,T2,T3,T4
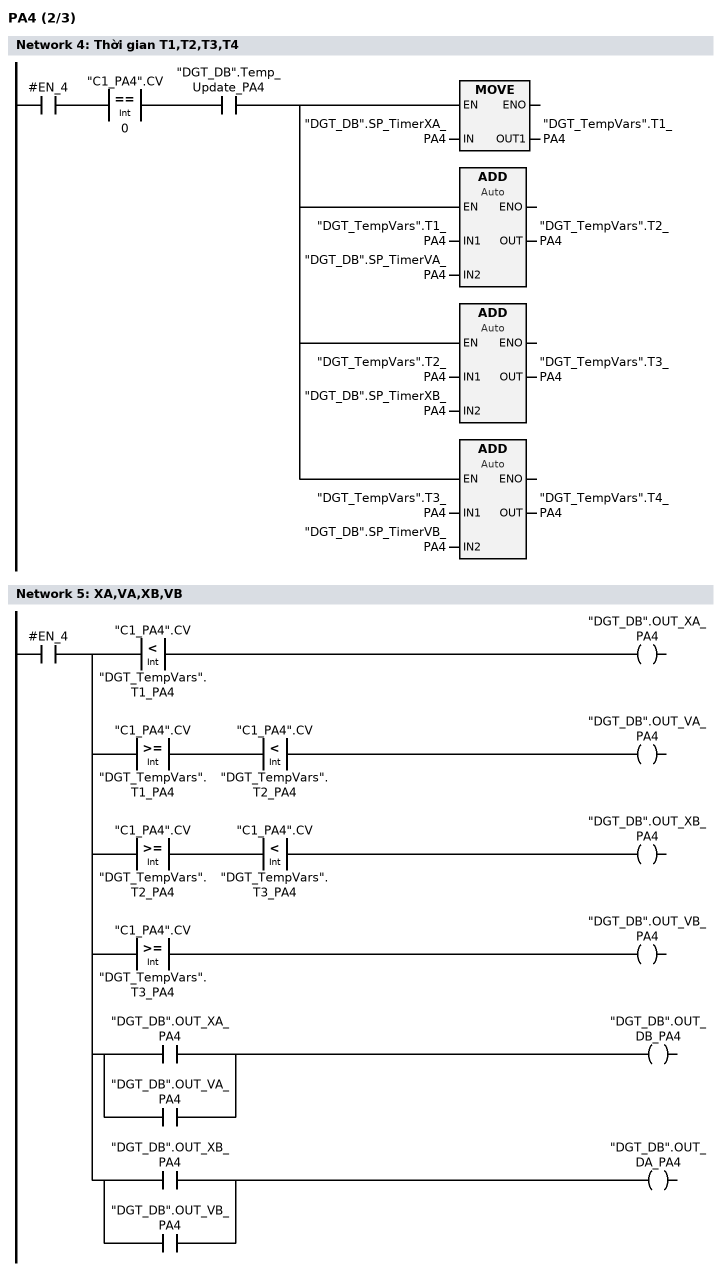
   RUNG wire#powerrail
      Contact( #EN_4 )
      { S7_Templates := "SrcType := Int" } EQ_Contact(in1 := "C1_PA4".CV, in2 := 0)
      Contact( "DGT_DB".Temp_Update_PA4 )
      wire#w1
      Move(in := "DGT_DB".SP_TimerXA_PA4, out1 => "DGT_TempVars".T1_PA4)
   END_RUNG
   RUNG wire#w1
      Add(in1 := "DGT_TempVars".T1_PA4, in2 := "DGT_DB".SP_TimerVA_PA4, out => "DGT_TempVars".T2_PA4)
   END_RUNG
   RUNG wire#w1
      Add(in1 := "DGT_TempVars".T2_PA4, in2 := "DGT_DB".SP_TimerXB_PA4, out => "DGT_TempVars".T3_PA4)
   END_RUNG
   RUNG wire#w1
      Add(in1 := "DGT_TempVars".T3_PA4, in2 := "DGT_DB".SP_TimerVB_PA4, out => "DGT_TempVars".T4_PA4)
   END_RUNG
   // the same network as SCL:
   IF #EN_4 AND ("C1_PA4".CV = 0) AND "DGT_DB".Temp_Update_PA4 THEN
       "DGT_TempVars".T1_PA4 := "DGT_DB".SP_TimerXA_PA4;
       "DGT_TempVars".T2_PA4 := "DGT_TempVars".T1_PA4 + "DGT_DB".SP_TimerVA_PA4;
       "DGT_TempVars".T3_PA4 := "DGT_TempVars".T2_PA4 + "DGT_DB".SP_TimerXB_PA4;
       "DGT_TempVars".T4_PA4 := "DGT_TempVars".T3_PA4 + "DGT_DB".SP_TimerVB_PA4;
   END_IF;
END_REGION

REGION Network 5: XA,VA,XB,VB
   RUNG wire#powerrail
      Contact( #EN_4 )
      wire#w1
      { S7_Templates := "SrcType := Int" } LT_Contact(in1 := "C1_PA4".CV, in2 := "DGT_TempVars".T1_PA4)
      Coil( "DGT_DB".OUT_XA_PA4 )
   END_RUNG
   RUNG wire#w1
      { S7_Templates := "SrcType := Int" } GE_Contact(in1 := "C1_PA4".CV, in2 := "DGT_TempVars".T1_PA4)
      { S7_Templates := "SrcType := Int" } LT_Contact(in1 := "C1_PA4".CV, in2 := "DGT_TempVars".T2_PA4)
      Coil( "DGT_DB".OUT_VA_PA4 )
   END_RUNG
   RUNG wire#w1
      { S7_Templates := "SrcType := Int" } GE_Contact(in1 := "C1_PA4".CV, in2 := "DGT_TempVars".T2_PA4)
      { S7_Templates := "SrcType := Int" } LT_Contact(in1 := "C1_PA4".CV, in2 := "DGT_TempVars".T3_PA4)
      Coil( "DGT_DB".OUT_XB_PA4 )
   END_RUNG
   RUNG wire#w1
      { S7_Templates := "SrcType := Int" } GE_Contact(in1 := "C1_PA4".CV, in2 := "DGT_TempVars".T3_PA4)
      Coil( "DGT_DB".OUT_VB_PA4 )
   END_RUNG
   RUNG wire#w1
      Contact( "DGT_DB".OUT_XA_PA4 )
      wire#w2
      Coil( "DGT_DB".OUT_DB_PA4 )
   END_RUNG
   RUNG wire#w1
      Contact( "DGT_DB".OUT_VA_PA4 )
   END_RUNG wire#w2
   RUNG wire#w1
      Contact( "DGT_DB".OUT_XB_PA4 )
      wire#w3
      Coil( "DGT_DB".OUT_DA_PA4 )
   END_RUNG
   RUNG wire#w1
      Contact( "DGT_DB".OUT_VB_PA4 )
   END_RUNG wire#w3
   // the same network as SCL:
   "DGT_DB".OUT_XA_PA4 := #EN_4 AND ("C1_PA4".CV < "DGT_TempVars".T1_PA4);
   "DGT_DB".OUT_VA_PA4 := #EN_4 AND ("C1_PA4".CV >= "DGT_TempVars".T1_PA4) AND ("C1_PA4".CV < "DGT_TempVars".T2_PA4);
   "DGT_DB".OUT_XB_PA4 := #EN_4 AND ("C1_PA4".CV >= "DGT_TempVars".T2_PA4) AND ("C1_PA4".CV < "DGT_TempVars".T3_PA4);
   "DGT_DB".OUT_VB_PA4 := #EN_4 AND ("C1_PA4".CV >= "DGT_TempVars".T3_PA4);
   "DGT_DB".OUT_DB_PA4 := #EN_4 AND ("DGT_DB".OUT_XA_PA4 OR "DGT_DB".OUT_VA_PA4);
   "DGT_DB".OUT_DA_PA4 := #EN_4 AND ("DGT_DB".OUT_XB_PA4 OR "DGT_DB".OUT_VB_PA4);
END_REGION

REGION Network 6
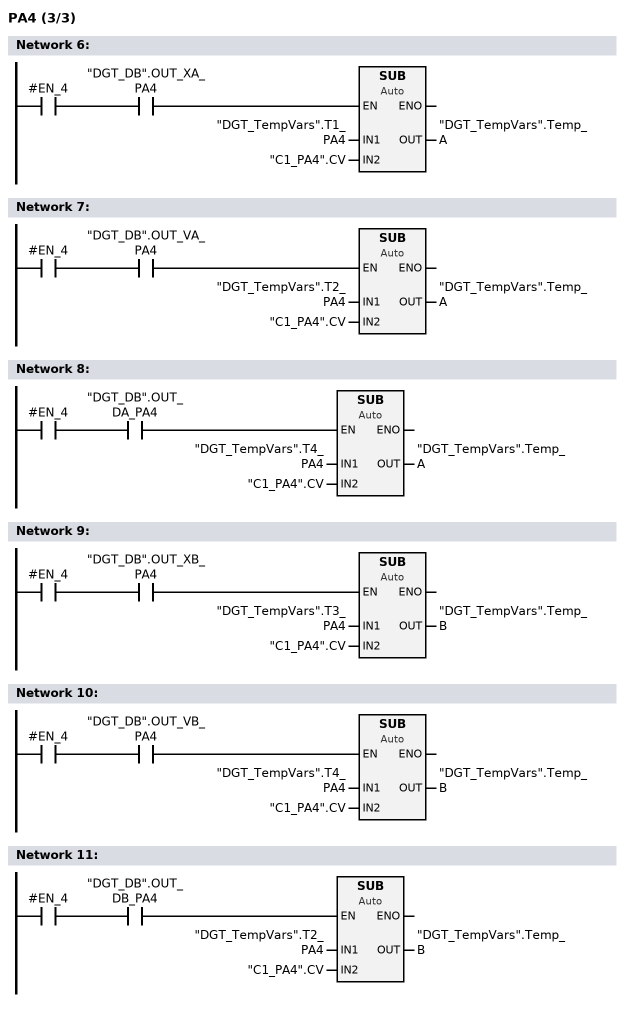
   RUNG wire#powerrail
      Contact( #EN_4 )
      Contact( "DGT_DB".OUT_XA_PA4 )
      Sub(in1 := "DGT_TempVars".T1_PA4, in2 := "C1_PA4".CV, out => "DGT_TempVars".Temp_A)
   END_RUNG
   // the same network as SCL:
   IF #EN_4 AND "DGT_DB".OUT_XA_PA4 THEN
       "DGT_TempVars".Temp_A := "DGT_TempVars".T1_PA4 - "C1_PA4".CV;
   END_IF;
END_REGION

REGION Network 7
   RUNG wire#powerrail
      Contact( #EN_4 )
      Contact( "DGT_DB".OUT_VA_PA4 )
      Sub(in1 := "DGT_TempVars".T2_PA4, in2 := "C1_PA4".CV, out => "DGT_TempVars".Temp_A)
   END_RUNG
   // the same network as SCL:
   IF #EN_4 AND "DGT_DB".OUT_VA_PA4 THEN
       "DGT_TempVars".Temp_A := "DGT_TempVars".T2_PA4 - "C1_PA4".CV;
   END_IF;
END_REGION

REGION Network 8
   RUNG wire#powerrail
      Contact( #EN_4 )
      Contact( "DGT_DB".OUT_DA_PA4 )
      Sub(in1 := "DGT_TempVars".T4_PA4, in2 := "C1_PA4".CV, out => "DGT_TempVars".Temp_A)
   END_RUNG
   // the same network as SCL:
   IF #EN_4 AND "DGT_DB".OUT_DA_PA4 THEN
       "DGT_TempVars".Temp_A := "DGT_TempVars".T4_PA4 - "C1_PA4".CV;
   END_IF;
END_REGION

REGION Network 9
   RUNG wire#powerrail
      Contact( #EN_4 )
      Contact( "DGT_DB".OUT_XB_PA4 )
      Sub(in1 := "DGT_TempVars".T3_PA4, in2 := "C1_PA4".CV, out => "DGT_TempVars".Temp_B)
   END_RUNG
   // the same network as SCL:
   IF #EN_4 AND "DGT_DB".OUT_XB_PA4 THEN
       "DGT_TempVars".Temp_B := "DGT_TempVars".T3_PA4 - "C1_PA4".CV;
   END_IF;
END_REGION

REGION Network 10
   RUNG wire#powerrail
      Contact( #EN_4 )
      Contact( "DGT_DB".OUT_VB_PA4 )
      Sub(in1 := "DGT_TempVars".T4_PA4, in2 := "C1_PA4".CV, out => "DGT_TempVars".Temp_B)
   END_RUNG
   // the same network as SCL:
   IF #EN_4 AND "DGT_DB".OUT_VB_PA4 THEN
       "DGT_TempVars".Temp_B := "DGT_TempVars".T4_PA4 - "C1_PA4".CV;
   END_IF;
END_REGION

REGION Network 11
   RUNG wire#powerrail
      Contact( #EN_4 )
      Contact( "DGT_DB".OUT_DB_PA4 )
      Sub(in1 := "DGT_TempVars".T2_PA4, in2 := "C1_PA4".CV, out => "DGT_TempVars".Temp_B)
   END_RUNG
   // the same network as SCL:
   IF #EN_4 AND "DGT_DB".OUT_DB_PA4 THEN
       "DGT_TempVars".Temp_B := "DGT_TempVars".T2_PA4 - "C1_PA4".CV;
   END_IF;
END_REGION
END_FUNCTION

ORGANIZATION_BLOCK "Main"   // OB1, LAD, ProgramCycle
TITLE = "Main Program Sweep (Cycle)"
{ S7_Optimized_Access := 'TRUE' }
VERSION : 0.1
   VAR_INPUT
      Initial_Call : Bool;   // Initial call of this OB
      Remanence : Bool;   // =True, if remanent data are available
   END_VAR
   VAR_TEMP   // added for the SCL form of the ladder/FBD networks
      _w1 : Bool;
   END_VAR
BEGIN

REGION Network 1
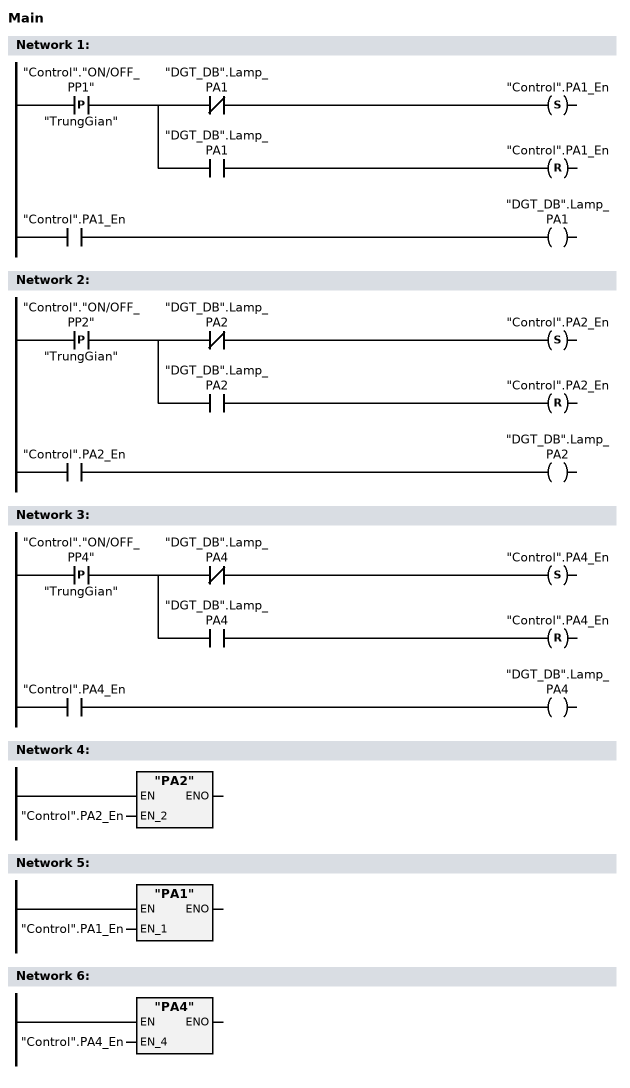
   RUNG wire#powerrail
      P_Contact(operand := "Control"."ON/OFF_PP1", bit := "TrungGian")
      wire#w1
      I_Contact( "DGT_DB".Lamp_PA1 )
      S_Coil( "Control".PA1_En )
   END_RUNG
   RUNG wire#w1
      Contact( "DGT_DB".Lamp_PA1 )
      R_Coil( "Control".PA1_En )
   END_RUNG
   RUNG wire#powerrail
      Contact( "Control".PA1_En )
      Coil( "DGT_DB".Lamp_PA1 )
   END_RUNG
   // the same network as SCL:
   #_w1 := "Control"."ON/OFF_PP1" AND NOT "TrungGian";   // rising edge of "Control"."ON/OFF_PP1"
   "TrungGian" := "Control"."ON/OFF_PP1";
   IF #_w1 AND NOT "DGT_DB".Lamp_PA1 THEN "Control".PA1_En := TRUE; END_IF;
   IF #_w1 AND "DGT_DB".Lamp_PA1 THEN "Control".PA1_En := FALSE; END_IF;
   "DGT_DB".Lamp_PA1 := "Control".PA1_En;
END_REGION

REGION Network 2
   RUNG wire#powerrail
      P_Contact(operand := "Control"."ON/OFF_PP2", bit := "TrungGian")
      wire#w1
      I_Contact( "DGT_DB".Lamp_PA2 )
      S_Coil( "Control".PA2_En )
   END_RUNG
   RUNG wire#w1
      Contact( "DGT_DB".Lamp_PA2 )
      R_Coil( "Control".PA2_En )
   END_RUNG
   RUNG wire#powerrail
      Contact( "Control".PA2_En )
      Coil( "DGT_DB".Lamp_PA2 )
   END_RUNG
   // the same network as SCL:
   #_w1 := "Control"."ON/OFF_PP2" AND NOT "TrungGian";   // rising edge of "Control"."ON/OFF_PP2"
   "TrungGian" := "Control"."ON/OFF_PP2";
   IF #_w1 AND NOT "DGT_DB".Lamp_PA2 THEN "Control".PA2_En := TRUE; END_IF;
   IF #_w1 AND "DGT_DB".Lamp_PA2 THEN "Control".PA2_En := FALSE; END_IF;
   "DGT_DB".Lamp_PA2 := "Control".PA2_En;
END_REGION

REGION Network 3
   RUNG wire#powerrail
      P_Contact(operand := "Control"."ON/OFF_PP4", bit := "TrungGian")
      wire#w1
      I_Contact( "DGT_DB".Lamp_PA4 )
      S_Coil( "Control".PA4_En )
   END_RUNG
   RUNG wire#w1
      Contact( "DGT_DB".Lamp_PA4 )
      R_Coil( "Control".PA4_En )
   END_RUNG
   RUNG wire#powerrail
      Contact( "Control".PA4_En )
      Coil( "DGT_DB".Lamp_PA4 )
   END_RUNG
   // the same network as SCL:
   #_w1 := "Control"."ON/OFF_PP4" AND NOT "TrungGian";   // rising edge of "Control"."ON/OFF_PP4"
   "TrungGian" := "Control"."ON/OFF_PP4";
   IF #_w1 AND NOT "DGT_DB".Lamp_PA4 THEN "Control".PA4_En := TRUE; END_IF;
   IF #_w1 AND "DGT_DB".Lamp_PA4 THEN "Control".PA4_En := FALSE; END_IF;
   "DGT_DB".Lamp_PA4 := "Control".PA4_En;
END_REGION

REGION Network 4
   RUNG wire#powerrail
      "PA2"(EN_2 := "Control".PA2_En)
   END_RUNG
   // the same network as SCL:
   "PA2"(EN_2 := "Control".PA2_En);
END_REGION

REGION Network 5
   RUNG wire#powerrail
      "PA1"(EN_1 := "Control".PA1_En)
   END_RUNG
   // the same network as SCL:
   "PA1"(EN_1 := "Control".PA1_En);
END_REGION

REGION Network 6
   RUNG wire#powerrail
      "PA4"(EN_4 := "Control".PA4_En)
   END_RUNG
   // the same network as SCL:
   "PA4"(EN_4 := "Control".PA4_En);
END_REGION
END_ORGANIZATION_BLOCK

(* ===== HMI "HMI_RT_1" =====
system functions are stored by id; their names below are inferred from use
connection "HMI_Connection_1": ETHERNET, SMART_S7_1200_OMS

HMI tags "Default tag table"
   "DGT_DB_SP_TimerXA" : Time = PLC DGT_DB.SP_TimerXA, 1 s
   "DGT_DB_SP_TimerVA" : Time = PLC DGT_DB.SP_TimerVA, 1 s
   "DGT_DB_SP_TimerXB" : Time = PLC DGT_DB.SP_TimerXB, 1 s
   "DGT_DB_SP_TimerVB" : Time = PLC DGT_DB.SP_TimerVB, 1 s
   "Timer_PP2_ET" : Time = PLC Timer_PP2.ET, 1 s
   "Control_PA2_En" : Bool = PLC Control.PA2_En, 1 s
   "Temp_A" : UInt = PLC DGT_TempVars.Temp_A AT %MD30, 1 s
   "Temp_B" : UInt = PLC DGT_TempVars.Temp_B AT %MD32, 1 s
   "DGT_TempVars_Temp_A" : UInt = PLC DGT_TempVars.Temp_A, 1 s
   "DGT_TempVars_Temp_B" : UInt = PLC DGT_TempVars.Temp_B, 1 s
   "DGT_TempVars_T1" : Time = PLC DGT_TempVars.T1, 1 s
   "DGT_TempVars_T2" : Time = PLC DGT_TempVars.T2, 1 s
   "DGT_TempVars_T3" : Time = PLC DGT_TempVars.T3, 1 s
   "DGT_TempVars_T4" : Time = PLC DGT_TempVars.T4, 1 s
   "DGT_DB_Lamp_PP2" : Bool = PLC DGT_DB.Lamp_PA2, 1 s
   "DGT_TempVars_Temp" : UInt = PLC DGT_TempVars.Temp, 1 s
   "DGT_DB_Update" : Bool = PLC DGT_DB.Update, 1 s
   "DGT_DB_Temp_Update" : Bool = PLC DGT_DB.Temp_Update, 1 s
   "DGT_DB_Cancel" : Bool = PLC DGT_DB.Cancel, 1 s
   "Control_PA1_En" : Bool = PLC Control.PA1_En, 1 s
   "DGT_TempVars_Temp_SP_XA" : Time = PLC DGT_TempVars.Temp_SP_XA, 1 s
   "DGT_TempVars_Temp_SP_VA" : Time = PLC DGT_TempVars.Temp_SP_VA, 1 s
   "DGT_TempVars_Temp_SP_XB" : Time = PLC DGT_TempVars.Temp_SP_XB, 1 s
   "DGT_TempVars_Temp_SP_VB" : Time = PLC DGT_TempVars.Temp_SP_VB, 1 s
   "Timer_PP1_ET" : Time = PLC Timer_PP1.ET, 1 s
   "DGT_DB_OUT_XA_PA2" : Bool = PLC DGT_DB.OUT_XA_PA2, 1 s
   "DGT_DB_OUT_VA_PA2" : Bool = PLC DGT_DB.OUT_VA_PA2, 1 s
   "DGT_DB_OUT_DA_PA2" : Bool = PLC DGT_DB.OUT_DA_PA2, 1 s
   "DGT_DB_OUT_XB_PA2" : Bool = PLC DGT_DB.OUT_XB_PA2, 1 s
   "DGT_DB_OUT_VB_PA2" : Bool = PLC DGT_DB.OUT_VB_PA2, 1 s
   "DGT_DB_OUT_DB_PA2" : Bool = PLC DGT_DB.OUT_DB_PA2, 1 s
   "DGT_DB_Lamp_PA1" : Bool = PLC DGT_DB.Lamp_PA1, 1 s
   "Control_ON/OFF_PP1" : Bool = PLC Control.ON/OFF_PP1, 1 s
   "Control_ON/OFF_PP2" : Bool = PLC Control.ON/OFF_PP2, 1 s
   "DGT_TempVars_T1_PA4" : Int = PLC DGT_TempVars.T1_PA4, 1 s
   "DGT_TempVars_T2_PA4" : Int = PLC DGT_TempVars.T2_PA4, 1 s
   "DGT_TempVars_T3_PA4" : Int = PLC DGT_TempVars.T3_PA4, 1 s
   "DGT_TempVars_T4_PA4" : Int = PLC DGT_TempVars.T4_PA4, 1 s
   "C1_PA4_CV" : Int = PLC C1_PA4.CV, 1 s
   "DGT_DB_OUT_XA_PA4" : Bool = PLC DGT_DB.OUT_XA_PA4, 1 s
   "DGT_DB_OUT_VA_PA4" : Bool = PLC DGT_DB.OUT_VA_PA4, 1 s
   "DGT_DB_OUT_DA_PA4" : Bool = PLC DGT_DB.OUT_DA_PA4, 1 s
   "DGT_DB_OUT_XB_PA4" : Bool = PLC DGT_DB.OUT_XB_PA4, 1 s
   "DGT_DB_OUT_VB_PA4" : Bool = PLC DGT_DB.OUT_VB_PA4, 1 s
   "DGT_DB_OUT_DB_PA4" : Bool = PLC DGT_DB.OUT_DB_PA4, 1 s
   "Control_ON/OFF_PP4" : Bool = PLC Control.ON/OFF_PP4, 1 s
   "DGT_DB_Lamp_PA4" : Bool = PLC DGT_DB.Lamp_PA4, 1 s
   "DGT_DB_SP_TimerXA_PA4" : Int = PLC DGT_DB.SP_TimerXA_PA4, 1 s
   "DGT_DB_SP_TimerVA_PA4" : Int = PLC DGT_DB.SP_TimerVA_PA4, 1 s
   "DGT_DB_SP_TimerXB_PA4" : Int = PLC DGT_DB.SP_TimerXB_PA4, 1 s
   "DGT_DB_SP_TimerVB_PA4" : Int = PLC DGT_DB.SP_TimerVB_PA4, 1 s
   "DGT_DB_Temp_Update_PA4" : Bool = PLC DGT_DB.Temp_Update_PA4, 1 s
   "DGT_DB_Update_PA4" : Bool = PLC DGT_DB.Update_PA4, 1 s
   "DGT_DB_OUT_XA" : Bool = PLC DGT_DB.OUT_XA, 1 s
   "DGT_DB_OUT_VA" : Bool = PLC DGT_DB.OUT_VA, 1 s
   "DGT_DB_OUT_DA" : Bool = PLC DGT_DB.OUT_DA, 1 s
   "DGT_DB_OUT_XB" : Bool = PLC DGT_DB.OUT_XB, 1 s
   "DGT_DB_OUT_VB" : Bool = PLC DGT_DB.OUT_VB, 1 s
   "DGT_DB_OUT_DB" : Bool = PLC DGT_DB.OUT_DB, 1 s
   "BCD_SEG_TEMPA_CHUC_SEG" : Byte = PLC BCD_SEG_TEMPA_CHUC.SEG, 1 s
   "BCD_SEG_TEMPA_DV_SEG" : Byte = PLC BCD_SEG_TEMPA_DV.SEG, 1 s
   "BCD_SEG_TEMPB_CHUC_SEG" : Byte = PLC BCD_SEG_TEMPB_CHUC.SEG, 1 s
   "BCD_SEG_TEMPB_DV_SEG" : Byte = PLC BCD_SEG_TEMPB_DV.SEG, 1 s

screen "Traffic_PA1" 800x480
   Circle "Circle_1" at 38,108 size 48x48
      Appearance <- "DGT_DB_OUT_DA"
   TextField "Text field_1" at 34,337 size 57x23; Text 'Side A'
   Circle "Circle_4" at 195,108 size 48x48
      Appearance <- "DGT_DB_OUT_DB"
   TextField "Text field_2" at 191,337 size 56x23; Text 'Side B'
   IOField "I/O field_6" at 23,36 size 83x41; FormatPattern 99
      ProcessValue <- "DGT_TempVars_Temp_A"
   IOField "I/O field_7" at 178,37 size 83x40; FormatPattern 99
      ProcessValue <- "DGT_TempVars_Temp_B"
   Circle "Circle_9" at 308,46 size 55x55
      Appearance <- "DGT_DB_Lamp_PA1"
   TextField "Text field_17" at 317,60 size 37x23; Text 'Run'
   Circle "Circle_10" at 308,106 size 55x55
      Appearance <- "DGT_DB_Temp_Update"
   TextField "Text field_19" at 309,122 size 51x20; Text 'Update'
   Button "Button_4" at 341,321 size 102x33; TextOff 'Start/Stop'
      on Press: SetBit("Control_ON/OFF_PP1")
      on Release: ResetBit("Control_ON/OFF_PP1")
   Button "Button_5" at 473,324 size 96x32; TextOff 'Update'
      on Release: ResetBit("DGT_DB_Update")
      on Press: SetBit("DGT_DB_Update")
   Button "Button_6" at 598,324 size 96x32; TextOff 'Cancel'
      on Release: ResetBit("DGT_DB_Cancel")
      on Press: SetBit("DGT_DB_Cancel")
   TextField "Text field_12" at 384,195 size 57x23; Text 'Side A'
   TextField "Text field_15" at 605,195 size 56x23; Text 'Side B'
   TextField "Text field_16" at 506,233 size 54x23; Text 'Green'
   TextField "Text field_20" at 506,271 size 60x23; Text 'Yellow'
   IOField "I/O field_12" at 366,225 size 107x32; FormatPattern s99999; Unit ms
      ProcessValue <- "DGT_DB_SP_TimerXA"
   IOField "I/O field_13" at 365,265 size 107x34; FormatPattern s99999; Unit ms
      ProcessValue <- "DGT_DB_SP_TimerVA"
   IOField "I/O field_14" at 569,223 size 114x36; FormatPattern s99999; Unit ms
      ProcessValue <- "DGT_DB_SP_TimerXB"
   IOField "I/O field_15" at 569,267 size 114x33; FormatPattern s99999; Unit ms
      ProcessValue <- "DGT_DB_SP_TimerVB"
   TextField "Text field_21" at 300,230 size 54x23; Text 'Green'
   TextField "Text field_22" at 300,270 size 60x23; Text 'Yellow'
   TextField "Text field_3" at 412,86 size 85x27; Text 'Running'
      Visibility <- "DGT_DB_Lamp_PA1"
   TextField "Text field_4" at 411,126 size 84x27; Text 'Stopped'
      Visibility <- "DGT_DB_Lamp_PA1"
   TextField "Text field_5" at 524,88 size 92x27; Text 'Updating'
      Visibility <- "DGT_DB_Temp_Update"
   TextField "Text field_7" at 523,127 size 85x27; Text 'Updated'
      Visibility <- "DGT_DB_Temp_Update"
   TextField "Text field_9" at 478,54 size 57x23; Text 'Status'
   IOField "I/O field_1" at 80,377 size 130x30; FormatPattern s9999999999
      ProcessValue <- "DGT_TempVars_Temp_SP_XA"
   IOField "I/O field_2" at 80,410 size 130x33; FormatPattern s9999999999
      ProcessValue <- "DGT_TempVars_Temp_SP_VA"
   IOField "I/O field_3" at 300,376 size 133x32; FormatPattern s9999999999
      ProcessValue <- "DGT_TempVars_Temp_SP_XB"
   IOField "I/O field_4" at 298,415 size 138x31; FormatPattern s9999999999
      ProcessValue <- "DGT_TempVars_Temp_SP_VB"
   IOField "I/O field_16" at 148,448 size 130x32; FormatPattern s9999999999
      ProcessValue <- "Timer_PP1_ET"
   TextField "Text field_6" at 261,7 size 286x27; Text 'Đèn Giao Thông Phương Án 1'
   Circle "Circle_2" at 38,246 size 48x48
      Appearance <- "DGT_DB_OUT_XA"
   Circle "Circle_3" at 38,175 size 48x48
      Appearance <- "DGT_DB_OUT_VA"
   Circle "Circle_5" at 193,240 size 48x48
      Appearance <- "DGT_DB_OUT_XB"
   Circle "Circle_6" at 193,175 size 48x48
      Appearance <- "DGT_DB_OUT_VB"
   TextField "Text field_8" at 113,453 size 26x23; Text 'ET'
   TextField "Text field_10" at 0,382 size 71x23; Text 'Green A'
   TextField "Text field_11" at 1,412 size 77x23; Text 'Yellow A'
   TextField "Text field_13" at 220,414 size 76x23; Text 'Yellow B'
   TextField "Text field_14" at 218,382 size 70x23; Text 'Green B'

screen "Traffic_PA2" 800x480
   Circle "Circle_1" at 39,151 size 48x48
      Appearance <- "DGT_DB_OUT_DA_PA2"
   Circle "Circle_2" at 39,217 size 48x48
      Appearance <- "DGT_DB_OUT_VA_PA2"
   Circle "Circle_3" at 39,284 size 48x48
      Appearance <- "DGT_DB_OUT_XA_PA2"
   TextField "Text field_1" at 35,344 size 57x23; Text 'Side A'
   Circle "Circle_4" at 196,148 size 48x48
      Appearance <- "DGT_DB_OUT_DB_PA2"
   Circle "Circle_5" at 196,214 size 48x48
      Appearance <- "DGT_DB_OUT_VB_PA2"
   Circle "Circle_6" at 196,281 size 48x48
      Appearance <- "DGT_DB_OUT_XB_PA2"
   TextField "Text field_2" at 192,344 size 56x23; Text 'Side B'
   IOField "I/O field_5" at 91,382 size 115x33; FormatPattern s99999; Unit ms
      ProcessValue <- "DGT_TempVars_T1"
   IOField "I/O field_8" at 93,415 size 113x34; FormatPattern s99999; Unit ms
      ProcessValue <- "DGT_TempVars_T2"
   IOField "I/O field_9" at 248,383 size 111x34; FormatPattern s99999; Unit ms
      ProcessValue <- "DGT_TempVars_T3"
   IOField "I/O field_10" at 248,417 size 112x31; FormatPattern s99999; Unit ms
      ProcessValue <- "DGT_TempVars_T4"
   IOField "I/O field_11" at 148,447 size 111x33; FormatPattern s99999; Unit ms
      ProcessValue <- "Timer_PP2_ET"
   TextField "Text field_6" at 56,386 size 26x23; Text 'T1'
   TextField "Text field_10" at 54,419 size 26x23; Text 'T2'
   TextField "Text field_11" at 222,386 size 26x23; Text 'T3'
   TextField "Text field_13" at 222,417 size 26x23; Text 'T4'
   TextField "Text field_14" at 107,449 size 26x23; Text 'ET'
   Circle "Circle_9" at 376,60 size 55x55
      Appearance <- "DGT_DB_Lamp_PP2"
   TextField "Text field_17" at 385,74 size 37x23; Text 'Run'
   Circle "Circle_10" at 376,120 size 55x55
      Appearance <- "DGT_DB_Temp_Update"
   TextField "Text field_19" at 377,136 size 51x20; Text 'Update'
   Button "Button_4" at 368,336 size 102x33; TextOff 'Start/Stop'
      on Release: ResetBit("Control_ON/OFF_PP2")
      on Press: SetBit("Control_ON/OFF_PP2")
   Button "Button_5" at 499,335 size 96x32; TextOff 'Update'
      on Release: ResetBit("DGT_DB_Update")
      on Press: SetBit("DGT_DB_Update")
   Button "Button_6" at 626,332 size 96x32; TextOff 'Cancel'
      on Release: ResetBit("DGT_DB_Cancel")
      on Press: SetBit("DGT_DB_Cancel")
   TextField "Text field_12" at 411,210 size 57x23; Text 'Side A'
   TextField "Text field_15" at 632,210 size 56x23; Text 'Side B'
   TextField "Text field_16" at 533,248 size 54x23; Text 'Green'
   TextField "Text field_20" at 533,286 size 60x23; Text 'Yellow'
   IOField "I/O field_12" at 393,240 size 107x32; FormatPattern s9999; Unit giây
      ProcessValue <- "DGT_DB_SP_TimerXA"
   IOField "I/O field_13" at 392,280 size 107x34; FormatPattern s9999; Unit giây
      ProcessValue <- "DGT_DB_SP_TimerVA"
   IOField "I/O field_14" at 596,238 size 114x36; FormatPattern s9999; Unit giây
      ProcessValue <- "DGT_DB_SP_TimerXB"
   IOField "I/O field_15" at 596,282 size 114x33; FormatPattern s9999; Unit giây
      ProcessValue <- "DGT_DB_SP_TimerVB"
   TextField "Text field_21" at 327,245 size 54x23; Text 'Green'
   TextField "Text field_22" at 327,285 size 60x23; Text 'Yellow'
   TextField "Text field_3" at 480,100 size 85x27; Text 'Running'
      Visibility <- "DGT_DB_Lamp_PP2"
   TextField "Text field_4" at 479,140 size 84x27; Text 'Stopped'
      Visibility <- "DGT_DB_Lamp_PP2"
   TextField "Text field_5" at 592,102 size 92x27; Text 'Updating'
      Visibility <- "DGT_DB_Temp_Update"
   TextField "Text field_7" at 591,141 size 85x27; Text 'Updated'
      Visibility <- "DGT_DB_Temp_Update"
   TextField "Text field_9" at 546,68 size 57x23; Text 'Status'
   TextField "Text field_18" at 9,405 size 36x23; Text 'PLC'
   Group "Group" at 16,34 size 100x93
   Group "Group_1" at 170,34 size 106x92
   TextField "Text field_23" at 387,12 size 250x27; Text 'Lập trình Đèn Giao Thông'
   Rectangle "Rectangle_7" at 21,34 size 38x8
      Appearance <- "BCD_SEG_TEMPA_CHUC_SEG"
   Rectangle "Rectangle_9" at 55,42 size 8x35
      Appearance <- "BCD_SEG_TEMPA_CHUC_SEG"
   Rectangle "Rectangle_10" at 16,42 size 8x35
      Appearance <- "BCD_SEG_TEMPA_CHUC_SEG"
   Rectangle "Rectangle_11" at 20,77 size 38x8
      Appearance <- "BCD_SEG_TEMPA_CHUC_SEG"
   Rectangle "Rectangle_12" at 54,84 size 8x35
      Appearance <- "BCD_SEG_TEMPA_CHUC_SEG"
   Rectangle "Rectangle_13" at 16,84 size 8x35
      Appearance <- "BCD_SEG_TEMPA_CHUC_SEG"
   Rectangle "Rectangle_14" at 21,119 size 38x8
      Appearance <- "BCD_SEG_TEMPA_CHUC_SEG"
   Rectangle "Rectangle_15" at 75,34 size 38x8
      Appearance <- "BCD_SEG_TEMPA_DV_SEG"
   Rectangle "Rectangle_16" at 108,42 size 8x35
      Appearance <- "BCD_SEG_TEMPA_DV_SEG"
   Rectangle "Rectangle_17" at 70,42 size 8x35
      Appearance <- "BCD_SEG_TEMPA_DV_SEG"
   Rectangle "Rectangle_18" at 74,77 size 38x8
      Appearance <- "BCD_SEG_TEMPA_DV_SEG"
   Rectangle "Rectangle_19" at 107,84 size 8x35
      Appearance <- "BCD_SEG_TEMPA_DV_SEG"
   Rectangle "Rectangle_20" at 70,84 size 8x35
      Appearance <- "BCD_SEG_TEMPA_DV_SEG"
   Rectangle "Rectangle_21" at 75,119 size 38x8
      Appearance <- "BCD_SEG_TEMPA_DV_SEG"
   Rectangle "Rectangle_22" at 175,34 size 40x8
      Appearance <- "BCD_SEG_TEMPB_CHUC_SEG"
   Rectangle "Rectangle_23" at 211,42 size 8x34
      Appearance <- "BCD_SEG_TEMPB_CHUC_SEG"
   Rectangle "Rectangle_24" at 170,42 size 8x34
      Appearance <- "BCD_SEG_TEMPB_CHUC_SEG"
   Rectangle "Rectangle_25" at 175,76 size 40x8
      Appearance <- "BCD_SEG_TEMPB_CHUC_SEG"
   Rectangle "Rectangle_26" at 210,84 size 8x34
      Appearance <- "BCD_SEG_TEMPB_CHUC_SEG"
   Rectangle "Rectangle_27" at 170,84 size 8x34
      Appearance <- "BCD_SEG_TEMPB_CHUC_SEG"
   Rectangle "Rectangle_28" at 175,118 size 40x8
      Appearance <- "BCD_SEG_TEMPB_CHUC_SEG"
   Rectangle "Rectangle_29" at 232,34 size 40x8
      Appearance <- "BCD_SEG_TEMPB_DV_SEG"
   Rectangle "Rectangle_30" at 268,42 size 8x34
      Appearance <- "BCD_SEG_TEMPB_DV_SEG"
   Rectangle "Rectangle_31" at 226,42 size 8x34
      Appearance <- "BCD_SEG_TEMPB_DV_SEG"
   Rectangle "Rectangle_32" at 231,76 size 40x8
      Appearance <- "BCD_SEG_TEMPB_DV_SEG"
   Rectangle "Rectangle_33" at 267,84 size 8x34
      Appearance <- "BCD_SEG_TEMPB_DV_SEG"
   Rectangle "Rectangle_34" at 226,84 size 8x34
      Appearance <- "BCD_SEG_TEMPB_DV_SEG"
   Rectangle "Rectangle_35" at 232,118 size 40x8
      Appearance <- "BCD_SEG_TEMPB_DV_SEG"

screen "Traffic_PA4" 800x480
   Circle "Circle_1" at 36,89 size 48x48
      Appearance <- "DGT_DB_OUT_DA_PA4"
   Circle "Circle_2" at 36,155 size 48x48
      Appearance <- "DGT_DB_OUT_VA_PA4"
   Circle "Circle_3" at 36,222 size 48x48
      Appearance <- "DGT_DB_OUT_XA_PA4"
   TextField "Text field_1" at 32,318 size 57x23; Text 'Side A'
   Circle "Circle_4" at 193,89 size 48x48
      Appearance <- "DGT_DB_OUT_DB_PA4"
   Circle "Circle_5" at 193,155 size 48x48
      Appearance <- "DGT_DB_OUT_VB_PA4"
   Circle "Circle_6" at 193,222 size 48x48
      Appearance <- "DGT_DB_OUT_XB_PA4"
   TextField "Text field_2" at 189,318 size 56x23; Text 'Side B'
   IOField "I/O field_6" at 21,17 size 83x41; FormatPattern 99
      ProcessValue <- "DGT_TempVars_Temp_A"
   IOField "I/O field_7" at 176,18 size 83x40; FormatPattern 99
      ProcessValue <- "DGT_TempVars_Temp_B"
   TextField "Text field_6" at 12,359 size 26x23; Text 'T1'
   TextField "Text field_10" at 9,404 size 26x23; Text 'T2'
   TextField "Text field_11" at 206,362 size 26x23; Text 'T3'
   TextField "Text field_13" at 203,408 size 26x23; Text 'T4'
   TextField "Text field_14" at 12,443 size 26x23; Text 'ET'
   Circle "Circle_9" at 306,27 size 55x55
      Appearance <- "DGT_DB_Lamp_PA4"
   TextField "Text field_17" at 315,41 size 37x23; Text 'Run'
   Circle "Circle_10" at 306,87 size 55x55
      Appearance <- "DGT_DB_Temp_Update_PA4"
   TextField "Text field_19" at 307,103 size 51x20; Text 'Update'
   Button "Button_4" at 339,302 size 102x33; TextOff 'Start/Stop'
      on Release: ResetBit("Control_ON/OFF_PP4")
      on Press: SetBit("Control_ON/OFF_PP4")
   Button "Button_5" at 471,305 size 96x32; TextOff 'Update'
      on Release: ResetBit("DGT_DB_Update_PA4")
      on Press: SetBit("DGT_DB_Update_PA4")
   Button "Button_6" at 596,305 size 96x32; TextOff 'Cancel'
      on Release: ResetBit("DGT_DB_Cancel")
      on Press: SetBit("DGT_DB_Cancel")
   TextField "Text field_12" at 382,176 size 57x23; Text 'Side A'
   TextField "Text field_15" at 603,176 size 56x23; Text 'Side B'
   TextField "Text field_16" at 504,214 size 54x23; Text 'Green'
   TextField "Text field_20" at 504,252 size 60x23; Text 'Yellow'
   IOField "I/O field_12" at 364,206 size 107x32; FormatPattern s99999; Unit s
      ProcessValue <- "DGT_DB_SP_TimerXA_PA4"
   IOField "I/O field_13" at 363,246 size 107x34; FormatPattern s99999; Unit s
      ProcessValue <- "DGT_DB_SP_TimerVA_PA4"
   IOField "I/O field_14" at 567,204 size 114x36; FormatPattern s99999; Unit s
      ProcessValue <- "DGT_DB_SP_TimerXB_PA4"
   IOField "I/O field_15" at 567,248 size 114x33; FormatPattern s99999; Unit s
      ProcessValue <- "DGT_DB_SP_TimerVB_PA4"
   TextField "Text field_21" at 298,211 size 54x23; Text 'Green'
   TextField "Text field_22" at 298,251 size 60x23; Text 'Yellow'
   TextField "Text field_3" at 410,67 size 85x27; Text 'Running'
      Visibility <- "DGT_DB_Lamp_PA4"
   TextField "Text field_4" at 409,107 size 84x27; Text 'Stopped'
      Visibility <- "DGT_DB_Lamp_PA4"
   TextField "Text field_5" at 522,69 size 92x27; Text 'Updating'
      Visibility <- "DGT_DB_Temp_Update_PA4"
   TextField "Text field_7" at 521,108 size 85x27; Text 'Updated'
      Visibility <- "DGT_DB_Temp_Update_PA4"
   TextField "Text field_9" at 476,35 size 57x23; Text 'Status'
   IOField "I/O field_1" at 45,359 size 96x32; FormatPattern s99999
      ProcessValue <- "DGT_TempVars_T1_PA4"
   IOField "I/O field_2" at 45,399 size 96x32; FormatPattern s99999
      ProcessValue <- "DGT_TempVars_T2_PA4"
   IOField "I/O field_3" at 240,362 size 96x32; FormatPattern s99999
      ProcessValue <- "DGT_TempVars_T3_PA4"
   IOField "I/O field_4" at 243,411 size 90x32; FormatPattern s99999
      ProcessValue <- "DGT_TempVars_T4_PA4"
   IOField "I/O field_5" at 46,443 size 96x32; FormatPattern s99999
      ProcessValue <- "C1_PA4_CV"
*)